   DATA[633,1] := 534.7403;
   DATA[633,2] := 2.0;
   DATA[633,3] := 2.0;
   DATA[633,4] := 262.1764;
   DATA[633,5] := 8.396116;
   DATA[633,6] := 327.7621;
   DATA[633,7] := 2.441675;
   DATA[633,8] := 2.0;
   DATA[633,9] := 2.0;
   DATA[633,10] := 2.0;
   DATA[633,11] := 19.68756;
   DATA[633,12] := 2.209653;
   DATA[633,13] := 985.4845;
   DATA[633,14] := 1.0;
   DATA[633,15] := 2.0;
   DATA[633,16] := 1.0;
   DATA[633,17] := 1.0;
   DATA[633,18] := 1.0;
   DATA[633,19] := 2.0;
   DATA[633,20] := 148.808;
   DATA[633,21] := 155.7806;
   DATA[633,22] := 1.719156;
   DATA[633,23] := 992.5147;
   DATA[633,24] := 2.0;
   DATA[633,25] := 2.0;
   DATA[633,26] := 7.87798;
   DATA[633,27] := 145.0141;
   DATA[633,28] := 263.1377;
   DATA[633,29] := 12.03538;
   DATA[633,30] := 1.731095;
   DATA[633,31] := 1.281542;
   DATA[633,32] := 0.7355248;
   DATA[633,33] := 0.3084265;
   DATA[633,34] := 2.0;
   DATA[633,35] := 250.8972;
   DATA[633,36] := 1.69801;
   DATA[633,37] := 189.6148;
   DATA[633,38] := 0.000128152;
   DATA[633,39] := 1.0;
   DATA[634,0] := 2.641002;
   DATA[634,1] := 534.6618;
   DATA[634,2] := 2.0;
   DATA[634,3] := 2.0;
   DATA[634,4] := 262.1764;
   DATA[634,5] := 8.396116;
   DATA[634,6] := 327.7621;
   DATA[634,7] := 2.44411;
   DATA[634,8] := 2.0;
   DATA[634,9] := 2.0;
   DATA[634,10] := 2.0;
   DATA[634,11] := 19.68756;
   DATA[634,12] := 2.21324;
   DATA[634,13] := 985.4845;
   DATA[634,14] := 1.0;
   DATA[634,15] := 2.0;
   DATA[634,16] := 1.0;
   DATA[634,17] := 1.0;
   DATA[634,18] := 1.0;
   DATA[634,19] := 2.0;
   DATA[634,20] := 148.808;
   DATA[634,21] := 155.7806;
   DATA[634,22] := 1.719156;
   DATA[634,23] := 992.7454;
   DATA[634,24] := 2.0;
   DATA[634,25] := 2.0;
   DATA[634,26] := 7.87798;
   DATA[634,27] := 144.9628;
   DATA[634,28] := 263.1377;
   DATA[634,29] := 12.03538;
   DATA[634,30] := 1.731095;
   DATA[634,31] := 1.281542;
   DATA[634,32] := 0.7355248;
   DATA[634,33] := 0.3080421;
   DATA[634,34] := 2.0;
   DATA[634,35] := 250.8972;
   DATA[634,36] := 1.69801;
   DATA[634,37] := 189.6148;
   DATA[634,38] := 0.000128152;
   DATA[634,39] := 1.0;
   DATA[635,0] := 2.657656;
   DATA[635,1] := 534.1516;
   DATA[635,2] := 2.0;
   DATA[635,3] := 2.0;
   DATA[635,4] := 262.1764;
   DATA[635,5] := 8.396116;
   DATA[635,6] := 327.7621;
   DATA[635,7] := 2.444366;
   DATA[635,8] := 2.0;
   DATA[635,9] := 2.0;
   DATA[635,10] := 2.0;
   DATA[635,11] := 19.68756;
   DATA[635,12] := 2.21324;
   DATA[635,13] := 985.4845;
   DATA[635,14] := 1.0;
   DATA[635,15] := 2.0;
   DATA[635,16] := 1.0;
   DATA[635,17] := 1.0;
   DATA[635,18] := 1.0;
   DATA[635,19] := 2.0;
   DATA[635,20] := 148.808;
   DATA[635,21] := 155.7806;
   DATA[635,22] := 1.717361;
   DATA[635,23] := 992.707;
   DATA[635,24] := 2.0;
   DATA[635,25] := 2.0;
   DATA[635,26] := 7.87798;
   DATA[635,27] := 144.9628;
   DATA[635,28] := 263.1377;
   DATA[635,29] := 12.03538;
   DATA[635,30] := 1.731095;
   DATA[635,31] := 1.282567;
   DATA[635,32] := 0.7355248;
   DATA[635,33] := 0.3066329;
   DATA[635,34] := 2.0;
   DATA[635,35] := 250.8972;
   DATA[635,36] := 1.69801;
   DATA[635,37] := 189.6148;
   DATA[635,38] := 0.000128152;
   DATA[635,39] := 1.0;
   DATA[636,0] := 2.663741;
   DATA[636,1] := 534.23;
   DATA[636,2] := 2.0;
   DATA[636,3] := 2.0;
   DATA[636,4] := 262.1764;
   DATA[636,5] := 8.396116;
   DATA[636,6] := 327.7621;
   DATA[636,7] := 2.444623;
   DATA[636,8] := 2.0;
   DATA[636,9] := 2.0;
   DATA[636,10] := 2.0;
   DATA[636,11] := 19.68756;
   DATA[636,12] := 2.21324;
   DATA[636,13] := 985.3644;
   DATA[636,14] := 1.0;
   DATA[636,15] := 2.0;
   DATA[636,16] := 1.0;
   DATA[636,17] := 1.0;
   DATA[636,18] := 1.0;
   DATA[636,19] := 2.0;
   DATA[636,20] := 148.808;
   DATA[636,21] := 155.7806;
   DATA[636,22] := 1.717361;
   DATA[636,23] := 992.6685;
   DATA[636,24] := 2.0;
   DATA[636,25] := 2.0;
   DATA[636,26] := 7.87798;
   DATA[636,27] := 144.9628;
   DATA[636,28] := 263.1377;
   DATA[636,29] := 12.03538;
   DATA[636,30] := 1.729172;
   DATA[636,31] := 1.289228;
   DATA[636,32] := 0.7355248;
   DATA[636,33] := 0.3081062;
   DATA[636,34] := 2.0;
   DATA[636,35] := 250.8972;
   DATA[636,36] := 1.69801;
   DATA[636,37] := 189.6148;
   DATA[636,38] := 0.000128152;
   DATA[636,39] := 1.0;
   DATA[637,0] := 2.660539;
   DATA[637,1] := 534.5048;
   DATA[637,2] := 2.0;
   DATA[637,3] := 2.0;
   DATA[637,4] := 262.1764;
   DATA[637,5] := 8.396116;
   DATA[637,6] := 327.7621;
   DATA[637,7] := 2.444623;
   DATA[637,8] := 2.0;
   DATA[637,9] := 2.0;
   DATA[637,10] := 2.0;
   DATA[637,11] := 19.67476;
   DATA[637,12] := 2.21324;
   DATA[637,13] := 985.6047;
   DATA[637,14] := 1.0;
   DATA[637,15] := 2.0;
   DATA[637,16] := 1.0;
   DATA[637,17] := 1.0;
   DATA[637,18] := 1.0;
   DATA[637,19] := 2.0;
   DATA[637,20] := 148.808;
   DATA[637,21] := 155.7806;
   DATA[637,22] := 1.717361;
   DATA[637,23] := 992.5916;
   DATA[637,24] := 2.0;
   DATA[637,25] := 2.0;
   DATA[637,26] := 7.87798;
   DATA[637,27] := 144.9628;
   DATA[637,28] := 263.1377;
   DATA[637,29] := 12.03538;
   DATA[637,30] := 1.729172;
   DATA[637,31] := 1.275266;
   DATA[637,32] := 0.7355248;
   DATA[637,33] := 0.3081062;
   DATA[637,34] := 2.0;
   DATA[637,35] := 250.8972;
   DATA[637,36] := 1.69801;
   DATA[637,37] := 189.6148;
   DATA[637,38] := 0.000128152;
   DATA[637,39] := 1.0;
   DATA[638,0] := 2.628511;
   DATA[638,1] := 534.9366;
   DATA[638,2] := 2.0;
   DATA[638,3] := 2.0;
   DATA[638,4] := 262.1764;
   DATA[638,5] := 8.396116;
   DATA[638,6] := 327.7621;
   DATA[638,7] := 2.443341;
   DATA[638,8] := 2.0;
   DATA[638,9] := 2.0;
   DATA[638,10] := 2.0;
   DATA[638,11] := 19.62354;
   DATA[638,12] := 2.211575;
   DATA[638,13] := 985.6848;
   DATA[638,14] := 1.0;
   DATA[638,15] := 2.0;
   DATA[638,16] := 1.0;
   DATA[638,17] := 1.0;
   DATA[638,18] := 1.0;
   DATA[638,19] := 2.0;
   DATA[638,20] := 148.808;
   DATA[638,21] := 155.7806;
   DATA[638,22] := 1.715567;
   DATA[638,23] := 992.5532;
   DATA[638,24] := 2.0;
   DATA[638,25] := 2.0;
   DATA[638,26] := 7.87798;
   DATA[638,27] := 144.9628;
   DATA[638,28] := 263.1377;
   DATA[638,29] := 12.34299;
   DATA[638,30] := 1.729172;
   DATA[638,31] := 1.261304;
   DATA[638,32] := 0.7355248;
   DATA[638,33] := 0.3081062;
   DATA[638,34] := 2.0;
   DATA[638,35] := 250.8972;
   DATA[638,36] := 1.69801;
   DATA[638,37] := 189.6148;
   DATA[638,38] := 0.000128152;
   DATA[638,39] := 1.0;
   DATA[639,0] := 2.622426;
   DATA[639,1] := 535.2114;
   DATA[639,2] := 2.0;
   DATA[639,3] := 2.0;
   DATA[639,4] := 262.1764;
   DATA[639,5] := 8.396116;
   DATA[639,6] := 327.7621;
   DATA[639,7] := 2.443341;
   DATA[639,8] := 2.0;
   DATA[639,9] := 2.0;
   DATA[639,10] := 2.0;
   DATA[639,11] := 19.60753;
   DATA[639,12] := 2.211447;
   DATA[639,13] := 985.8851;
   DATA[639,14] := 1.0;
   DATA[639,15] := 2.0;
   DATA[639,16] := 1.0;
   DATA[639,17] := 1.0;
   DATA[639,18] := 1.0;
   DATA[639,19] := 2.0;
   DATA[639,20] := 148.808;
   DATA[639,21] := 155.7806;
   DATA[639,22] := 1.715567;
   DATA[639,23] := 992.5532;
   DATA[639,24] := 2.0;
   DATA[639,25] := 2.0;
   DATA[639,26] := 7.87798;
   DATA[639,27] := 144.9628;
   DATA[639,28] := 263.1377;
   DATA[639,29] := 12.34299;
   DATA[639,30] := 1.729172;
   DATA[639,31] := 1.261944;
   DATA[639,32] := 0.7355248;
   DATA[639,33] := 0.3081062;
   DATA[639,34] := 2.0;
   DATA[639,35] := 250.8972;
   DATA[639,36] := 1.617916;
   DATA[639,37] := 189.6148;
   DATA[639,38] := 0.000128152;
   DATA[639,39] := 1.0;
   DATA[640,0] := 2.616981;
   DATA[640,1] := 535.2114;
   DATA[640,2] := 2.0;
   DATA[640,3] := 2.0;
   DATA[640,4] := 262.1764;
   DATA[640,5] := 8.395155;
   DATA[640,6] := 327.7621;
   DATA[640,7] := 2.443341;
   DATA[640,8] := 2.0;
   DATA[640,9] := 2.0;
   DATA[640,10] := 2.0;
   DATA[640,11] := 19.57872;
   DATA[640,12] := 2.211447;
   DATA[640,13] := 985.7649;
   DATA[640,14] := 1.0;
   DATA[640,15] := 2.0;
   DATA[640,16] := 1.0;
   DATA[640,17] := 1.0;
   DATA[640,18] := 1.0;
   DATA[640,19] := 2.0;
   DATA[640,20] := 148.808;
   DATA[640,21] := 155.7806;
   DATA[640,22] := 1.715567;
   DATA[640,23] := 992.7839;
   DATA[640,24] := 2.0;
   DATA[640,25] := 2.0;
   DATA[640,26] := 7.87798;
   DATA[640,27] := 144.9628;
   DATA[640,28] := 263.1377;
   DATA[640,29] := 12.34299;
   DATA[640,30] := 1.729172;
   DATA[640,31] := 1.280902;
   DATA[640,32] := 0.7355248;
   DATA[640,33] := 0.3081062;
   DATA[640,34] := 2.0;
   DATA[640,35] := 250.8972;
   DATA[640,36] := 1.617916;
   DATA[640,37] := 189.6148;
   DATA[640,38] := 0.000128152;
   DATA[640,39] := 1.0;
   DATA[641,0] := 2.601287;
   DATA[641,1] := 535.3291;
   DATA[641,2] := 2.0;
   DATA[641,3] := 2.0;
   DATA[641,4] := 262.1764;
   DATA[641,5] := 8.395155;
   DATA[641,6] := 327.7621;
   DATA[641,7] := 2.443341;
   DATA[641,8] := 2.0;
   DATA[641,9] := 2.0;
   DATA[641,10] := 2.0;
   DATA[641,11] := 19.5275;
   DATA[641,12] := 2.211447;
   DATA[641,13] := 986.0052;
   DATA[641,14] := 1.0;
   DATA[641,15] := 2.0;
   DATA[641,16] := 1.0;
   DATA[641,17] := 1.0;
   DATA[641,18] := 1.0;
   DATA[641,19] := 2.0;
   DATA[641,20] := 148.808;
   DATA[641,21] := 155.7806;
   DATA[641,22] := 1.715567;
   DATA[641,23] := 992.8608;
   DATA[641,24] := 2.0;
   DATA[641,25] := 2.0;
   DATA[641,26] := 7.87798;
   DATA[641,27] := 144.9628;
   DATA[641,28] := 263.1377;
   DATA[641,29] := 12.15073;
   DATA[641,30] := 1.729172;
   DATA[641,31] := 1.28167;
   DATA[641,32] := 0.7355248;
   DATA[641,33] := 0.3081062;
   DATA[641,34] := 2.0;
   DATA[641,35] := 250.8972;
   DATA[641,36] := 1.617916;
   DATA[641,37] := 189.6148;
   DATA[641,38] := 0.000128152;
   DATA[641,39] := 1.0;
   DATA[642,0] := 2.585914;
   DATA[642,1] := 535.4469;
   DATA[642,2] := 2.0;
   DATA[642,3] := 2.0;
   DATA[642,4] := 262.1764;
   DATA[642,5] := 8.395155;
   DATA[642,6] := 327.7621;
   DATA[642,7] := 2.440393;
   DATA[642,8] := 2.0;
   DATA[642,9] := 2.0;
   DATA[642,10] := 2.0;
   DATA[642,11] := 19.5275;
   DATA[642,12] := 2.211447;
   DATA[642,13] := 986.0853;
   DATA[642,14] := 1.0;
   DATA[642,15] := 2.0;
   DATA[642,16] := 1.0;
   DATA[642,17] := 1.0;
   DATA[642,18] := 1.0;
   DATA[642,19] := 2.0;
   DATA[642,20] := 148.808;
   DATA[642,21] := 155.7806;
   DATA[642,22] := 1.715567;
   DATA[642,23] := 992.9761;
   DATA[642,24] := 2.0;
   DATA[642,25] := 2.0;
   DATA[642,26] := 7.878942;
   DATA[642,27] := 144.9628;
   DATA[642,28] := 263.1377;
   DATA[642,29] := 12.03538;
   DATA[642,30] := 1.729172;
   DATA[642,31] := 1.28167;
   DATA[642,32] := 0.7339884;
   DATA[642,33] := 0.3084905;
   DATA[642,34] := 2.0;
   DATA[642,35] := 250.8972;
   DATA[642,36] := 1.617916;
   DATA[642,37] := 189.6148;
   DATA[642,38] := 0.000128152;
   DATA[642,39] := 1.0;
   DATA[643,0] := 2.564456;
   DATA[643,1] := 535.8394;
   DATA[643,2] := 2.0;
   DATA[643,3] := 2.0;
   DATA[643,4] := 262.1764;
   DATA[643,5] := 8.395155;
   DATA[643,6] := 327.7621;
   DATA[643,7] := 2.439753;
   DATA[643,8] := 2.0;
   DATA[643,9] := 2.0;
   DATA[643,10] := 2.0;
   DATA[643,11] := 19.5275;
   DATA[643,12] := 2.211447;
   DATA[643,13] := 986.0853;
   DATA[643,14] := 1.0;
   DATA[643,15] := 2.0;
   DATA[643,16] := 1.0;
   DATA[643,17] := 1.0;
   DATA[643,18] := 1.0;
   DATA[643,19] := 2.0;
   DATA[643,20] := 148.808;
   DATA[643,21] := 155.7806;
   DATA[643,22] := 1.715567;
   DATA[643,23] := 993.053;
   DATA[643,24] := 2.0;
   DATA[643,25] := 2.0;
   DATA[643,26] := 7.878942;
   DATA[643,27] := 144.9628;
   DATA[643,28] := 263.1377;
   DATA[643,29] := 12.03538;
   DATA[643,30] := 1.730838;
   DATA[643,31] := 1.277956;
   DATA[643,32] := 0.7339884;
   DATA[643,33] := 0.3084905;
   DATA[643,34] := 2.0;
   DATA[643,35] := 250.8972;
   DATA[643,36] := 1.617916;
   DATA[643,37] := 189.6148;
   DATA[643,38] := 0.000128152;
   DATA[643,39] := 1.0;
   DATA[644,0] := 2.548762;
   DATA[644,1] := 535.6431;
   DATA[644,2] := 2.0;
   DATA[644,3] := 2.0;
   DATA[644,4] := 262.1764;
   DATA[644,5] := 8.395155;
   DATA[644,6] := 327.7621;
   DATA[644,7] := 2.439753;
   DATA[644,8] := 2.0;
   DATA[644,9] := 2.0;
   DATA[644,10] := 2.0;
   DATA[644,11] := 19.59793;
   DATA[644,12] := 2.210166;
   DATA[644,13] := 986.2856;
   DATA[644,14] := 1.0;
   DATA[644,15] := 2.0;
   DATA[644,16] := 1.0;
   DATA[644,17] := 1.0;
   DATA[644,18] := 1.0;
   DATA[644,19] := 2.0;
   DATA[644,20] := 148.808;
   DATA[644,21] := 155.7806;
   DATA[644,22] := 1.715567;
   DATA[644,23] := 993.0915;
   DATA[644,24] := 2.0;
   DATA[644,25] := 2.0;
   DATA[644,26] := 7.878942;
   DATA[644,27] := 144.9628;
   DATA[644,28] := 263.1697;
   DATA[644,29] := 12.03538;
   DATA[644,30] := 1.730838;
   DATA[644,31] := 1.275266;
   DATA[644,32] := 0.7360369;
   DATA[644,33] := 0.3084905;
   DATA[644,34] := 2.0;
   DATA[644,35] := 250.8011;
   DATA[644,36] := 1.762086;
   DATA[644,37] := 189.5668;
   DATA[644,38] := 0.000128152;
   DATA[644,39] := 1.0;
   DATA[645,0] := 2.533068;
   DATA[645,1] := 535.2506;
   DATA[645,2] := 2.0;
   DATA[645,3] := 2.0;
   DATA[645,4] := 262.1764;
   DATA[645,5] := 8.395155;
   DATA[645,6] := 327.7621;
   DATA[645,7] := 2.439753;
   DATA[645,8] := 2.0;
   DATA[645,9] := 2.0;
   DATA[645,10] := 2.0;
   DATA[645,11] := 19.62674;
   DATA[645,12] := 2.210166;
   DATA[645,13] := 986.6461;
   DATA[645,14] := 1.0;
   DATA[645,15] := 2.0;
   DATA[645,16] := 1.0;
   DATA[645,17] := 1.0;
   DATA[645,18] := 1.0;
   DATA[645,19] := 2.0;
   DATA[645,20] := 148.808;
   DATA[645,21] := 155.7806;
   DATA[645,22] := 1.714798;
   DATA[645,23] := 992.9761;
   DATA[645,24] := 2.0;
   DATA[645,25] := 2.0;
   DATA[645,26] := 7.878942;
   DATA[645,27] := 144.9628;
   DATA[645,28] := 263.4261;
   DATA[645,29] := 12.03538;
   DATA[645,30] := 1.730838;
   DATA[645,31] := 1.289484;
   DATA[645,32] := 0.7360369;
   DATA[645,33] := 0.3074016;
   DATA[645,34] := 2.0;
   DATA[645,35] := 250.6569;
   DATA[645,36] := 1.762086;
   DATA[645,37] := 189.5347;
   DATA[645,38] := 0.000128152;
   DATA[645,39] := 1.0;
   DATA[646,0] := 2.517695;
   DATA[646,1] := 534.8973;
   DATA[646,2] := 2.0;
   DATA[646,3] := 2.0;
   DATA[646,4] := 262.1764;
   DATA[646,5] := 8.395155;
   DATA[646,6] := 327.7621;
   DATA[646,7] := 2.439753;
   DATA[646,8] := 2.0;
   DATA[646,9] := 2.0;
   DATA[646,10] := 2.0;
   DATA[646,11] := 19.62674;
   DATA[646,12] := 2.210166;
   DATA[646,13] := 987.0466;
   DATA[646,14] := 1.0;
   DATA[646,15] := 2.0;
   DATA[646,16] := 1.0;
   DATA[646,17] := 1.0;
   DATA[646,18] := 1.0;
   DATA[646,19] := 2.0;
   DATA[646,20] := 148.808;
   DATA[646,21] := 155.7806;
   DATA[646,22] := 1.714542;
   DATA[646,23] := 993.053;
   DATA[646,24] := 2.0;
   DATA[646,25] := 2.0;
   DATA[646,26] := 7.878942;
   DATA[646,27] := 145.1166;
   DATA[646,28] := 263.4261;
   DATA[646,29] := 12.03538;
   DATA[646,30] := 1.727634;
   DATA[646,31] := 1.300756;
   DATA[646,32] := 0.7360369;
   DATA[646,33] := 0.3068251;
   DATA[646,34] := 2.0;
   DATA[646,35] := 250.6569;
   DATA[646,36] := 1.762086;
   DATA[646,37] := 189.5027;
   DATA[646,38] := 0.000128152;
   DATA[646,39] := 1.0;
   DATA[647,0] := 2.498799;
   DATA[647,1] := 534.6226;
   DATA[647,2] := 2.0;
   DATA[647,3] := 2.0;
   DATA[647,4] := 262.1764;
   DATA[647,5] := 8.395155;
   DATA[647,6] := 327.7621;
   DATA[647,7] := 2.439753;
   DATA[647,8] := 2.0;
   DATA[647,9] := 2.0;
   DATA[647,10] := 2.0;
   DATA[647,11] := 19.62674;
   DATA[647,12] := 2.211447;
   DATA[647,13] := 987.4471;
   DATA[647,14] := 1.0;
   DATA[647,15] := 2.0;
   DATA[647,16] := 1.0;
   DATA[647,17] := 1.0;
   DATA[647,18] := 1.0;
   DATA[647,19] := 2.0;
   DATA[647,20] := 148.808;
   DATA[647,21] := 155.7806;
   DATA[647,22] := 1.714542;
   DATA[647,23] := 992.8992;
   DATA[647,24] := 2.0;
   DATA[647,25] := 2.0;
   DATA[647,26] := 7.878942;
   DATA[647,27] := 145.1166;
   DATA[647,28] := 263.4261;
   DATA[647,29] := 12.03538;
   DATA[647,30] := 1.727634;
   DATA[647,31] := 1.297554;
   DATA[647,32] := 0.7360369;
   DATA[647,33] := 0.3068251;
   DATA[647,34] := 2.0;
   DATA[647,35] := 250.6569;
   DATA[647,36] := 1.601897;
   DATA[647,37] := 189.3745;
   DATA[647,38] := 0.000128152;
   DATA[647,39] := 1.0;
   DATA[648,0] := 2.483426;
   DATA[648,1] := 534.3085;
   DATA[648,2] := 2.0;
   DATA[648,3] := 2.0;
   DATA[648,4] := 262.1764;
   DATA[648,5] := 8.395155;
   DATA[648,6] := 327.7621;
   DATA[648,7] := 2.439753;
   DATA[648,8] := 2.0;
   DATA[648,9] := 2.0;
   DATA[648,10] := 2.0;
   DATA[648,11] := 19.66835;
   DATA[648,12] := 2.211447;
   DATA[648,13] := 987.0867;
   DATA[648,14] := 1.0;
   DATA[648,15] := 2.0;
   DATA[648,16] := 1.0;
   DATA[648,17] := 1.0;
   DATA[648,18] := 1.0;
   DATA[648,19] := 2.0;
   DATA[648,20] := 148.808;
   DATA[648,21] := 155.7806;
   DATA[648,22] := 1.715824;
   DATA[648,23] := 993.2453;
   DATA[648,24] := 2.0;
   DATA[648,25] := 2.0;
   DATA[648,26] := 7.878942;
   DATA[648,27] := 145.1166;
   DATA[648,28] := 263.4261;
   DATA[648,29] := 12.03538;
   DATA[648,30] := 1.727634;
   DATA[648,31] := 1.291918;
   DATA[648,32] := 0.7346286;
   DATA[648,33] := 0.3068251;
   DATA[648,34] := 2.0;
   DATA[648,35] := 250.6569;
   DATA[648,36] := 1.601897;
   DATA[648,37] := 189.3745;
   DATA[648,38] := 0.000128152;
   DATA[648,39] := 1.0;
   DATA[649,0] := 2.463248;
   DATA[649,1] := 534.6226;
   DATA[649,2] := 2.0;
   DATA[649,3] := 2.0;
   DATA[649,4] := 262.1764;
   DATA[649,5] := 8.395155;
   DATA[649,6] := 327.7621;
   DATA[649,7] := 2.439753;
   DATA[649,8] := 2.0;
   DATA[649,9] := 2.0;
   DATA[649,10] := 2.0;
   DATA[649,11] := 19.57552;
   DATA[649,12] := 2.211447;
   DATA[649,13] := 987.2068;
   DATA[649,14] := 1.0;
   DATA[649,15] := 2.0;
   DATA[649,16] := 1.0;
   DATA[649,17] := 1.0;
   DATA[649,18] := 1.0;
   DATA[649,19] := 2.0;
   DATA[649,20] := 148.808;
   DATA[649,21] := 155.7806;
   DATA[649,22] := 1.716849;
   DATA[649,23] := 993.2453;
   DATA[649,24] := 2.0;
   DATA[649,25] := 2.0;
   DATA[649,26] := 7.878942;
   DATA[649,27] := 145.1166;
   DATA[649,28] := 263.1697;
   DATA[649,29] := 12.03538;
   DATA[649,30] := 1.727634;
   DATA[649,31] := 1.281927;
   DATA[649,32] := 0.7346286;
   DATA[649,33] := 0.3066329;
   DATA[649,34] := 2.0;
   DATA[649,35] := 250.6569;
   DATA[649,36] := 1.601897;
   DATA[649,37] := 189.3745;
   DATA[649,38] := 0.000128152;
   DATA[649,39] := 1.0;
   DATA[650,0] := 2.463248;
   DATA[650,1] := 534.6226;
   DATA[650,2] := 2.0;
   DATA[650,3] := 2.0;
   DATA[650,4] := 262.1764;
   DATA[650,5] := 8.395155;
   DATA[650,6] := 327.7621;
   DATA[650,7] := 2.439753;
   DATA[650,8] := 2.0;
   DATA[650,9] := 2.0;
   DATA[650,10] := 2.0;
   DATA[650,11] := 19.57552;
   DATA[650,12] := 2.211447;
   DATA[650,13] := 987.2068;
   DATA[650,14] := 1.0;
   DATA[650,15] := 2.0;
   DATA[650,16] := 1.0;
   DATA[650,17] := 1.0;
   DATA[650,18] := 1.0;
   DATA[650,19] := 2.0;
   DATA[650,20] := 148.808;
   DATA[650,21] := 155.7806;
   DATA[650,22] := 1.716849;
   DATA[650,23] := 993.2453;
   DATA[650,24] := 2.0;
   DATA[650,25] := 2.0;
   DATA[650,26] := 7.878942;
   DATA[650,27] := 145.1166;
   DATA[650,28] := 263.1697;
   DATA[650,29] := 12.03538;
   DATA[650,30] := 1.727634;
   DATA[650,31] := 1.281927;
   DATA[650,32] := 0.7346286;
   DATA[650,33] := 0.3066329;
   DATA[650,34] := 2.0;
   DATA[650,35] := 250.6569;
   DATA[650,36] := 1.601897;
   DATA[650,37] := 189.3745;
   DATA[650,38] := 0.000128152;
   DATA[650,39] := 1.0;
   DATA[651,0] := 2.447234;
   DATA[651,1] := 534.701;
   DATA[651,2] := 2.0;
   DATA[651,3] := 2.0;
   DATA[651,4] := 262.1764;
   DATA[651,5] := 8.395155;
   DATA[651,6] := 327.7621;
   DATA[651,7] := 2.439753;
   DATA[651,8] := 2.0;
   DATA[651,9] := 2.0;
   DATA[651,10] := 2.0;
   DATA[651,11] := 19.57552;
   DATA[651,12] := 2.212856;
   DATA[651,13] := 987.0065;
   DATA[651,14] := 1.0;
   DATA[651,15] := 2.0;
   DATA[651,16] := 1.0;
   DATA[651,17] := 1.0;
   DATA[651,18] := 1.0;
   DATA[651,19] := 2.0;
   DATA[651,20] := 148.808;
   DATA[651,21] := 155.7806;
   DATA[651,22] := 1.717361;
   DATA[651,23] := 993.1684;
   DATA[651,24] := 2.0;
   DATA[651,25] := 2.0;
   DATA[651,26] := 7.878942;
   DATA[651,27] := 145.1166;
   DATA[651,28] := 263.1697;
   DATA[651,29] := 12.03538;
   DATA[651,30] := 1.727634;
   DATA[651,31] := 1.281158;
   DATA[651,32] := 0.7346286;
   DATA[651,33] := 0.3066329;
   DATA[651,34] := 2.0;
   DATA[651,35] := 250.8331;
   DATA[651,36] := 1.601897;
   DATA[651,37] := 189.6629;
   DATA[651,38] := 0.000128152;
   DATA[651,39] := 1.0;
   DATA[652,0] := 2.431861;
   DATA[652,1] := 535.9179;
   DATA[652,2] := 2.0;
   DATA[652,3] := 2.0;
   DATA[652,4] := 262.1764;
   DATA[652,5] := 8.395155;
   DATA[652,6] := 327.7621;
   DATA[652,7] := 2.44206;
   DATA[652,8] := 2.0;
   DATA[652,9] := 2.0;
   DATA[652,10] := 2.0;
   DATA[652,11] := 19.57552;
   DATA[652,12] := 2.212856;
   DATA[652,13] := 987.0466;
   DATA[652,14] := 1.0;
   DATA[652,15] := 2.0;
   DATA[652,16] := 1.0;
   DATA[652,17] := 1.0;
   DATA[652,18] := 1.0;
   DATA[652,19] := 2.0;
   DATA[652,20] := 148.808;
   DATA[652,21] := 155.7806;
   DATA[652,22] := 1.719284;
   DATA[652,23] := 993.3607;
   DATA[652,24] := 2.0;
   DATA[652,25] := 2.0;
   DATA[652,26] := 7.878942;
   DATA[652,27] := 145.1166;
   DATA[652,28] := 263.1697;
   DATA[652,29] := 12.03538;
   DATA[652,30] := 1.725968;
   DATA[652,31] := 1.289356;
   DATA[652,32] := 0.7361649;
   DATA[652,33] := 0.3066329;
   DATA[652,34] := 2.0;
   DATA[652,35] := 250.8331;
   DATA[652,36] := 1.601897;
   DATA[652,37] := 189.6629;
   DATA[652,38] := 0.000128152;
   DATA[652,39] := 1.0;
   DATA[653,0] := 2.428979;
   DATA[653,1] := 537.017;
   DATA[653,2] := 2.0;
   DATA[653,3] := 2.0;
   DATA[653,4] := 262.1764;
   DATA[653,5] := 8.395155;
   DATA[653,6] := 327.7621;
   DATA[653,7] := 2.44206;
   DATA[653,8] := 2.0;
   DATA[653,9] := 2.0;
   DATA[653,10] := 2.0;
   DATA[653,11] := 19.67155;
   DATA[653,12] := 2.212856;
   DATA[653,13] := 987.9678;
   DATA[653,14] := 1.0;
   DATA[653,15] := 2.0;
   DATA[653,16] := 1.0;
   DATA[653,17] := 1.0;
   DATA[653,18] := 1.0;
   DATA[653,19] := 2.0;
   DATA[653,20] := 148.808;
   DATA[653,21] := 155.7806;
   DATA[653,22] := 1.719412;
   DATA[653,23] := 993.8605;
   DATA[653,24] := 2.0;
   DATA[653,25] := 2.0;
   DATA[653,26] := 7.878942;
   DATA[653,27] := 145.0141;
   DATA[653,28] := 263.1697;
   DATA[653,29] := 12.03538;
   DATA[653,30] := 1.725968;
   DATA[653,31] := 1.296273;
   DATA[653,32] := 0.7361649;
   DATA[653,33] := 0.3066329;
   DATA[653,34] := 2.0;
   DATA[653,35] := 250.9613;
   DATA[653,36] := 1.601897;
   DATA[653,37] := 189.6629;
   DATA[653,38] := 0.000128152;
   DATA[653,39] := 1.0;
   DATA[654,0] := 2.431861;
   DATA[654,1] := 537.488;
   DATA[654,2] := 2.0;
   DATA[654,3] := 2.0;
   DATA[654,4] := 262.1764;
   DATA[654,5] := 8.395155;
   DATA[654,6] := 327.7621;
   DATA[654,7] := 2.44206;
   DATA[654,8] := 2.0;
   DATA[654,9] := 2.0;
   DATA[654,10] := 2.0;
   DATA[654,11] := 19.67155;
   DATA[654,12] := 2.212856;
   DATA[654,13] := 987.7676;
   DATA[654,14] := 1.0;
   DATA[654,15] := 2.0;
   DATA[654,16] := 1.0;
   DATA[654,17] := 1.0;
   DATA[654,18] := 1.0;
   DATA[654,19] := 2.0;
   DATA[654,20] := 148.808;
   DATA[654,21] := 155.7806;
   DATA[654,22] := 1.719412;
   DATA[654,23] := 994.1297;
   DATA[654,24] := 2.0;
   DATA[654,25] := 2.0;
   DATA[654,26] := 7.878942;
   DATA[654,27] := 144.9628;
   DATA[654,28] := 263.1697;
   DATA[654,29] := 12.03538;
   DATA[654,30] := 1.729557;
   DATA[654,31] := 1.308825;
   DATA[654,32] := 0.7361649;
   DATA[654,33] := 0.3066329;
   DATA[654,34] := 2.0;
   DATA[654,35] := 250.9613;
   DATA[654,36] := 1.601897;
   DATA[654,37] := 189.6629;
   DATA[654,38] := 0.000128152;
   DATA[654,39] := 1.0;
   DATA[655,0] := 2.475419;
   DATA[655,1] := 537.8806;
   DATA[655,2] := 2.0;
   DATA[655,3] := 2.0;
   DATA[655,4] := 262.1764;
   DATA[655,5] := 8.395155;
   DATA[655,6] := 327.7621;
   DATA[655,7] := 2.44206;
   DATA[655,8] := 2.0;
   DATA[655,9] := 2.0;
   DATA[655,10] := 2.0;
   DATA[655,11] := 19.67155;
   DATA[655,12] := 2.21119;
   DATA[655,13] := 987.8878;
   DATA[655,14] := 1.0;
   DATA[655,15] := 2.0;
   DATA[655,16] := 1.0;
   DATA[655,17] := 1.0;
   DATA[655,18] := 1.0;
   DATA[655,19] := 2.0;
   DATA[655,20] := 148.808;
   DATA[655,21] := 155.7806;
   DATA[655,22] := 1.719412;
   DATA[655,23] := 994.5142;
   DATA[655,24] := 2.0;
   DATA[655,25] := 2.0;
   DATA[655,26] := 7.878942;
   DATA[655,27] := 144.9628;
   DATA[655,28] := 263.1697;
   DATA[655,29] := 12.03538;
   DATA[655,30] := 1.730454;
   DATA[655,31] := 1.305495;
   DATA[655,32] := 0.7342445;
   DATA[655,33] := 0.3066329;
   DATA[655,34] := 2.0;
   DATA[655,35] := 251.1215;
   DATA[655,36] := 1.746067;
   DATA[655,37] := 189.6629;
   DATA[655,38] := 0.000128152;
   DATA[655,39] := 1.0;
   DATA[656,0] := 2.526022;
   DATA[656,1] := 538.1553;
   DATA[656,2] := 2.0;
   DATA[656,3] := 2.0;
   DATA[656,4] := 262.1764;
   DATA[656,5] := 8.395155;
   DATA[656,6] := 327.7621;
   DATA[656,7] := 2.44206;
   DATA[656,8] := 2.0;
   DATA[656,9] := 2.0;
   DATA[656,10] := 2.0;
   DATA[656,11] := 19.62994;
   DATA[656,12] := 2.210806;
   DATA[656,13] := 988.048;
   DATA[656,14] := 1.0;
   DATA[656,15] := 2.0;
   DATA[656,16] := 1.0;
   DATA[656,17] := 1.0;
   DATA[656,18] := 1.0;
   DATA[656,19] := 2.0;
   DATA[656,20] := 148.808;
   DATA[656,21] := 155.7806;
   DATA[656,22] := 1.719412;
   DATA[656,23] := 994.5142;
   DATA[656,24] := 2.0;
   DATA[656,25] := 2.0;
   DATA[656,26] := 7.878942;
   DATA[656,27] := 144.9628;
   DATA[656,28] := 263.1697;
   DATA[656,29] := 12.03538;
   DATA[656,30] := 1.73071;
   DATA[656,31] := 1.311387;
   DATA[656,32] := 0.7342445;
   DATA[656,33] := 0.3066329;
   DATA[656,34] := 2.0;
   DATA[656,35] := 251.1375;
   DATA[656,36] := 1.746067;
   DATA[656,37] := 189.759;
   DATA[656,38] := 0.000128152;
   DATA[656,39] := 1.0;
   DATA[657,0] := 2.556449;
   DATA[657,1] := 537.8413;
   DATA[657,2] := 2.0;
   DATA[657,3] := 2.0;
   DATA[657,4] := 262.1764;
   DATA[657,5] := 8.395155;
   DATA[657,6] := 327.7621;
   DATA[657,7] := 2.44206;
   DATA[657,8] := 2.0;
   DATA[657,9] := 2.0;
   DATA[657,10] := 2.0;
   DATA[657,11] := 19.62994;
   DATA[657,12] := 2.210806;
   DATA[657,13] := 988.2883;
   DATA[657,14] := 1.0;
   DATA[657,15] := 2.0;
   DATA[657,16] := 1.0;
   DATA[657,17] := 1.0;
   DATA[657,18] := 1.0;
   DATA[657,19] := 2.0;
   DATA[657,20] := 148.808;
   DATA[657,21] := 155.7806;
   DATA[657,22] := 1.719412;
   DATA[657,23] := 995.0141;
   DATA[657,24] := 2.0;
   DATA[657,25] := 2.0;
   DATA[657,26] := 7.878942;
   DATA[657,27] := 144.9628;
   DATA[657,28] := 263.1697;
   DATA[657,29] := 12.07383;
   DATA[657,30] := 1.73071;
   DATA[657,31] := 1.307929;
   DATA[657,32] := 0.7342445;
   DATA[657,33] := 0.3066329;
   DATA[657,34] := 2.0;
   DATA[657,35] := 251.3779;
   DATA[657,36] := 1.746067;
   DATA[657,37] := 189.8071;
   DATA[657,38] := 0.000128152;
   DATA[657,39] := 1.0;
   DATA[658,0] := 2.597764;
   DATA[658,1] := 537.6058;
   DATA[658,2] := 2.0;
   DATA[658,3] := 2.0;
   DATA[658,4] := 262.1764;
   DATA[658,5] := 8.395155;
   DATA[658,6] := 327.7621;
   DATA[658,7] := 2.44206;
   DATA[658,8] := 2.0;
   DATA[658,9] := 2.0;
   DATA[658,10] := 2.0;
   DATA[658,11] := 19.62994;
   DATA[658,12] := 2.210806;
   DATA[658,13] := 988.4084;
   DATA[658,14] := 1.0;
   DATA[658,15] := 2.0;
   DATA[658,16] := 1.0;
   DATA[658,17] := 1.0;
   DATA[658,18] := 1.0;
   DATA[658,19] := 2.0;
   DATA[658,20] := 148.808;
   DATA[658,21] := 155.7806;
   DATA[658,22] := 1.719412;
   DATA[658,23] := 995.0526;
   DATA[658,24] := 2.0;
   DATA[658,25] := 2.0;
   DATA[658,26] := 7.878942;
   DATA[658,27] := 144.9628;
   DATA[658,28] := 263.1697;
   DATA[658,29] := 12.07383;
   DATA[658,30] := 1.73212;
   DATA[658,31] := 1.30178;
   DATA[658,32] := 0.7352687;
   DATA[658,33] := 0.3066329;
   DATA[658,34] := 2.0;
   DATA[658,35] := 251.3779;
   DATA[658,36] := 1.746067;
   DATA[658,37] := 189.9353;
   DATA[658,38] := 0.000128152;
   DATA[658,39] := 1.0;
   DATA[659,0] := 2.626589;
   DATA[659,1] := 537.4095;
   DATA[659,2] := 2.0;
   DATA[659,3] := 2.0;
   DATA[659,4] := 262.1764;
   DATA[659,5] := 8.395155;
   DATA[659,6] := 327.7621;
   DATA[659,7] := 2.440906;
   DATA[659,8] := 2.0;
   DATA[659,9] := 2.0;
   DATA[659,10] := 2.0;
   DATA[659,11] := 19.62994;
   DATA[659,12] := 2.210806;
   DATA[659,13] := 988.4485;
   DATA[659,14] := 1.0;
   DATA[659,15] := 2.0;
   DATA[659,16] := 1.0;
   DATA[659,17] := 1.0;
   DATA[659,18] := 1.0;
   DATA[659,19] := 2.0;
   DATA[659,20] := 148.808;
   DATA[659,21] := 155.7806;
   DATA[659,22] := 1.719412;
   DATA[659,23] := 995.3986;
   DATA[659,24] := 2.0;
   DATA[659,25] := 2.0;
   DATA[659,26] := 7.878942;
   DATA[659,27] := 144.9628;
   DATA[659,28] := 263.2658;
   DATA[659,29] := 12.07383;
   DATA[659,30] := 1.73212;
   DATA[659,31] := 1.293711;
   DATA[659,32] := 0.7359089;
   DATA[659,33] := 0.3066329;
   DATA[659,34] := 2.0;
   DATA[659,35] := 251.3779;
   DATA[659,36] := 1.746067;
   DATA[659,37] := 189.9353;
   DATA[659,38] := 0.000128152;
   DATA[659,39] := 1.0;
   DATA[660,0] := 2.657016;
   DATA[660,1] := 537.3702;
   DATA[660,2] := 2.0;
   DATA[660,3] := 2.0;
   DATA[660,4] := 262.1764;
   DATA[660,5] := 8.395155;
   DATA[660,6] := 327.7621;
   DATA[660,7] := 2.440906;
   DATA[660,8] := 2.0;
   DATA[660,9] := 2.0;
   DATA[660,10] := 2.0;
   DATA[660,11] := 19.62994;
   DATA[660,12] := 2.210806;
   DATA[660,13] := 988.2883;
   DATA[660,14] := 1.0;
   DATA[660,15] := 2.0;
   DATA[660,16] := 1.0;
   DATA[660,17] := 1.0;
   DATA[660,18] := 1.0;
   DATA[660,19] := 2.0;
   DATA[660,20] := 148.808;
   DATA[660,21] := 155.7806;
   DATA[660,22] := 1.72159;
   DATA[660,23] := 995.4755;
   DATA[660,24] := 2.0;
   DATA[660,25] := 2.0;
   DATA[660,26] := 7.878942;
   DATA[660,27] := 144.9628;
   DATA[660,28] := 263.362;
   DATA[660,29] := 12.07383;
   DATA[660,30] := 1.73212;
   DATA[660,31] := 1.28372;
   DATA[660,32] := 0.7359089;
   DATA[660,33] := 0.3066329;
   DATA[660,34] := 2.0;
   DATA[660,35] := 251.2016;
   DATA[660,36] := 1.746067;
   DATA[660,37] := 189.9353;
   DATA[660,38] := 0.000128152;
   DATA[660,39] := 1.0;
   DATA[661,0] := 2.667585;
   DATA[661,1] := 537.0562;
   DATA[661,2] := 2.0;
   DATA[661,3] := 2.0;
   DATA[661,4] := 262.1764;
   DATA[661,5] := 8.395155;
   DATA[661,6] := 327.7621;
   DATA[661,7] := 2.440906;
   DATA[661,8] := 2.0;
   DATA[661,9] := 2.0;
   DATA[661,10] := 2.0;
   DATA[661,11] := 19.65555;
   DATA[661,12] := 2.209525;
   DATA[661,13] := 988.5687;
   DATA[661,14] := 1.0;
   DATA[661,15] := 2.0;
   DATA[661,16] := 1.0;
   DATA[661,17] := 1.0;
   DATA[661,18] := 1.0;
   DATA[661,19] := 2.0;
   DATA[661,20] := 148.808;
   DATA[661,21] := 155.7806;
   DATA[661,22] := 1.721975;
   DATA[661,23] := 995.6293;
   DATA[661,24] := 2.0;
   DATA[661,25] := 2.0;
   DATA[661,26] := 7.878942;
   DATA[661,27] := 144.9628;
   DATA[661,28] := 263.362;
   DATA[661,29] := 12.07383;
   DATA[661,30] := 1.73212;
   DATA[661,31] := 1.272192;
   DATA[661,32] := 0.7359089;
   DATA[661,33] := 0.3066329;
   DATA[661,34] := 2.0;
   DATA[661,35] := 251.0574;
   DATA[661,36] := 1.746067;
   DATA[661,37] := 189.9353;
   DATA[661,38] := 0.000128152;
   DATA[661,39] := 1.0;
   DATA[662,0] := 2.657976;
   DATA[662,1] := 537.0955;
   DATA[662,2] := 2.0;
   DATA[662,3] := 2.0;
   DATA[662,4] := 262.1764;
   DATA[662,5] := 8.395155;
   DATA[662,6] := 327.7621;
   DATA[662,7] := 2.443725;
   DATA[662,8] := 2.0;
   DATA[662,9] := 2.0;
   DATA[662,10] := 2.0;
   DATA[662,11] := 19.65555;
   DATA[662,12] := 2.209525;
   DATA[662,13] := 988.4485;
   DATA[662,14] := 1.0;
   DATA[662,15] := 2.0;
   DATA[662,16] := 1.0;
   DATA[662,17] := 1.0;
   DATA[662,18] := 1.0;
   DATA[662,19] := 2.0;
   DATA[662,20] := 148.808;
   DATA[662,21] := 155.7806;
   DATA[662,22] := 1.721975;
   DATA[662,23] := 996.0139;
   DATA[662,24] := 2.0;
   DATA[662,25] := 2.0;
   DATA[662,26] := 7.878942;
   DATA[662,27] := 144.9628;
   DATA[662,28] := 263.362;
   DATA[662,29] := 12.07383;
   DATA[662,30] := 1.73212;
   DATA[662,31] := 1.271295;
   DATA[662,32] := 0.7359089;
   DATA[662,33] := 0.3066329;
   DATA[662,34] := 2.0;
   DATA[662,35] := 251.0574;
   DATA[662,36] := 1.746067;
   DATA[662,37] := 189.9353;
   DATA[662,38] := 0.000128152;
   DATA[662,39] := 1.0;
   DATA[663,0] := 2.631393;
   DATA[663,1] := 537.2133;
   DATA[663,2] := 2.0;
   DATA[663,3] := 2.0;
   DATA[663,4] := 262.1764;
   DATA[663,5] := 8.395155;
   DATA[663,6] := 327.7621;
   DATA[663,7] := 2.444366;
   DATA[663,8] := 2.0;
   DATA[663,9] := 2.0;
   DATA[663,10] := 2.0;
   DATA[663,11] := 19.65555;
   DATA[663,12] := 2.213368;
   DATA[663,13] := 988.048;
   DATA[663,14] := 1.0;
   DATA[663,15] := 2.0;
   DATA[663,16] := 1.0;
   DATA[663,17] := 1.0;
   DATA[663,18] := 1.0;
   DATA[663,19] := 2.0;
   DATA[663,20] := 148.808;
   DATA[663,21] := 155.7806;
   DATA[663,22] := 1.720565;
   DATA[663,23] := 995.9754;
   DATA[663,24] := 2.0;
   DATA[663,25] := 2.0;
   DATA[663,26] := 7.878942;
   DATA[663,27] := 144.9628;
   DATA[663,28] := 263.362;
   DATA[663,29] := 12.07383;
   DATA[663,30] := 1.73212;
   DATA[663,31] := 1.262073;
   DATA[663,32] := 0.7357808;
   DATA[663,33] := 0.3066329;
   DATA[663,34] := 2.0;
   DATA[663,35] := 251.0574;
   DATA[663,36] := 1.746067;
   DATA[663,37] := 189.759;
   DATA[663,38] := 0.000128152;
   DATA[663,39] := 1.0;
   DATA[664,0] := 2.620824;
   DATA[664,1] := 537.0955;
   DATA[664,2] := 2.0;
   DATA[664,3] := 2.0;
   DATA[664,4] := 262.1764;
   DATA[664,5] := 8.395155;
   DATA[664,6] := 327.7621;
   DATA[664,7] := 2.445007;
   DATA[664,8] := 2.0;
   DATA[664,9] := 2.0;
   DATA[664,10] := 2.0;
   DATA[664,11] := 19.70357;
   DATA[664,12] := 2.211831;
   DATA[664,13] := 987.8878;
   DATA[664,14] := 1.0;
   DATA[664,15] := 2.0;
   DATA[664,16] := 1.0;
   DATA[664,17] := 1.0;
   DATA[664,18] := 1.0;
   DATA[664,19] := 2.0;
   DATA[664,20] := 148.808;
   DATA[664,21] := 155.6524;
   DATA[664,22] := 1.719027;
   DATA[664,23] := 996.2446;
   DATA[664,24] := 2.0;
   DATA[664,25] := 2.0;
   DATA[664,26] := 7.878942;
   DATA[664,27] := 144.9628;
   DATA[664,28] := 263.362;
   DATA[664,29] := 12.07383;
   DATA[664,30] := 1.73212;
   DATA[664,31] := 1.254771;
   DATA[664,32] := 0.7357808;
   DATA[664,33] := 0.3066329;
   DATA[664,34] := 2.0;
   DATA[664,35] := 251.0574;
   DATA[664,36] := 1.746067;
   DATA[664,37] := 189.743;
   DATA[664,38] := 0.000128152;
   DATA[664,39] := 1.0;
   DATA[665,0] := 2.620824;
   DATA[665,1] := 537.2917;
   DATA[665,2] := 2.0;
   DATA[665,3] := 2.0;
   DATA[665,4] := 262.1764;
   DATA[665,5] := 8.395155;
   DATA[665,6] := 327.7621;
   DATA[665,7] := 2.445007;
   DATA[665,8] := 2.0;
   DATA[665,9] := 2.0;
   DATA[665,10] := 2.0;
   DATA[665,11] := 19.70357;
   DATA[665,12] := 2.209909;
   DATA[665,13] := 988.088;
   DATA[665,14] := 1.0;
   DATA[665,15] := 2.0;
   DATA[665,16] := 1.0;
   DATA[665,17] := 1.0;
   DATA[665,18] := 1.0;
   DATA[665,19] := 2.0;
   DATA[665,20] := 148.808;
   DATA[665,21] := 155.5242;
   DATA[665,22] := 1.719027;
   DATA[665,23] := 995.937;
   DATA[665,24] := 2.0;
   DATA[665,25] := 2.0;
   DATA[665,26] := 7.878942;
   DATA[665,27] := 144.9628;
   DATA[665,28] := 263.2979;
   DATA[665,29] := 12.07383;
   DATA[665,30] := 1.73212;
   DATA[665,31] := 1.255796;
   DATA[665,32] := 0.7357808;
   DATA[665,33] := 0.3066329;
   DATA[665,34] := 2.0;
   DATA[665,35] := 251.0574;
   DATA[665,36] := 1.601897;
   DATA[665,37] := 189.743;
   DATA[665,38] := 0.000128152;
   DATA[665,39] := 1.0;
   DATA[666,0] := 2.613778;
   DATA[666,1] := 536.6245;
   DATA[666,2] := 2.0;
   DATA[666,3] := 2.0;
   DATA[666,4] := 262.1764;
   DATA[666,5] := 8.395155;
   DATA[666,6] := 327.7621;
   DATA[666,7] := 2.445007;
   DATA[666,8] := 2.0;
   DATA[666,9] := 2.0;
   DATA[666,10] := 2.0;
   DATA[666,11] := 19.70357;
   DATA[666,12] := 2.209909;
   DATA[666,13] := 987.9678;
   DATA[666,14] := 1.0;
   DATA[666,15] := 2.0;
   DATA[666,16] := 1.0;
   DATA[666,17] := 1.0;
   DATA[666,18] := 1.0;
   DATA[666,19] := 2.0;
   DATA[666,20] := 148.808;
   DATA[666,21] := 155.5242;
   DATA[666,22] := 1.718643;
   DATA[666,23] := 996.0139;
   DATA[666,24] := 2.0;
   DATA[666,25] := 2.0;
   DATA[666,26] := 7.878942;
   DATA[666,27] := 144.9628;
   DATA[666,28] := 263.2658;
   DATA[666,29] := 12.07383;
   DATA[666,30] := 1.73212;
   DATA[666,31] := 1.261432;
   DATA[666,32] := 0.7357808;
   DATA[666,33] := 0.3066329;
   DATA[666,34] := 2.0;
   DATA[666,35] := 251.0574;
   DATA[666,36] := 1.601897;
   DATA[666,37] := 189.743;
   DATA[666,38] := 0.000128152;
   DATA[666,39] := 1.0;
   DATA[667,0] := 2.598725;
   DATA[667,1] := 535.8787;
   DATA[667,2] := 2.0;
   DATA[667,3] := 2.0;
   DATA[667,4] := 262.1764;
   DATA[667,5] := 8.395155;
   DATA[667,6] := 327.7621;
   DATA[667,7] := 2.445007;
   DATA[667,8] := 2.0;
   DATA[667,9] := 2.0;
   DATA[667,10] := 2.0;
   DATA[667,11] := 19.75799;
   DATA[667,12] := 2.211575;
   DATA[667,13] := 988.0079;
   DATA[667,14] := 1.0;
   DATA[667,15] := 2.0;
   DATA[667,16] := 1.0;
   DATA[667,17] := 1.0;
   DATA[667,18] := 1.0;
   DATA[667,19] := 2.0;
   DATA[667,20] := 148.808;
   DATA[667,21] := 155.5242;
   DATA[667,22] := 1.718643;
   DATA[667,23] := 996.2446;
   DATA[667,24] := 2.0;
   DATA[667,25] := 2.0;
   DATA[667,26] := 7.878942;
   DATA[667,27] := 144.9628;
   DATA[667,28] := 263.2658;
   DATA[667,29] := 12.07383;
   DATA[667,30] := 1.729557;
   DATA[667,31] := 1.270783;
   DATA[667,32] := 0.7357808;
   DATA[667,33] := 0.3066329;
   DATA[667,34] := 2.0;
   DATA[667,35] := 251.0574;
   DATA[667,36] := 1.601897;
   DATA[667,37] := 189.743;
   DATA[667,38] := 0.000128152;
   DATA[667,39] := 1.0;
   DATA[668,0] := 2.58111;
   DATA[668,1] := 535.2899;
   DATA[668,2] := 2.0;
   DATA[668,3] := 2.0;
   DATA[668,4] := 262.1764;
   DATA[668,5] := 8.395155;
   DATA[668,6] := 327.7621;
   DATA[668,7] := 2.443341;
   DATA[668,8] := 2.0;
   DATA[668,9] := 2.0;
   DATA[668,10] := 2.0;
   DATA[668,11] := 19.77079;
   DATA[668,12] := 2.212856;
   DATA[668,13] := 987.8076;
   DATA[668,14] := 1.0;
   DATA[668,15] := 2.0;
   DATA[668,16] := 1.0;
   DATA[668,17] := 1.0;
   DATA[668,18] := 1.0;
   DATA[668,19] := 2.0;
   DATA[668,20] := 148.808;
   DATA[668,21] := 155.5242;
   DATA[668,22] := 1.718643;
   DATA[668,23] := 996.2061;
   DATA[668,24] := 2.0;
   DATA[668,25] := 2.0;
   DATA[668,26] := 7.878942;
   DATA[668,27] := 144.9628;
   DATA[668,28] := 263.2658;
   DATA[668,29] := 12.07383;
   DATA[668,30] := 1.729557;
   DATA[668,31] := 1.288843;
   DATA[668,32] := 0.7357808;
   DATA[668,33] := 0.3066329;
   DATA[668,34] := 2.0;
   DATA[668,35] := 250.9933;
   DATA[668,36] := 1.665972;
   DATA[668,37] := 189.743;
   DATA[668,38] := 0.000128152;
   DATA[668,39] := 1.0;
   DATA[669,0] := 2.564135;
   DATA[669,1] := 534.701;
   DATA[669,2] := 2.0;
   DATA[669,3] := 2.0;
   DATA[669,4] := 262.1764;
   DATA[669,5] := 8.395155;
   DATA[669,6] := 327.7621;
   DATA[669,7] := 2.443341;
   DATA[669,8] := 2.0;
   DATA[669,9] := 2.0;
   DATA[669,10] := 2.0;
   DATA[669,11] := 19.77079;
   DATA[669,12] := 2.212856;
   DATA[669,13] := 987.4071;
   DATA[669,14] := 1.0;
   DATA[669,15] := 2.0;
   DATA[669,16] := 1.0;
   DATA[669,17] := 1.0;
   DATA[669,18] := 1.0;
   DATA[669,19] := 2.0;
   DATA[669,20] := 148.808;
   DATA[669,21] := 155.5242;
   DATA[669,22] := 1.718643;
   DATA[669,23] := 995.9754;
   DATA[669,24] := 2.0;
   DATA[669,25] := 2.0;
   DATA[669,26] := 7.878942;
   DATA[669,27] := 144.9628;
   DATA[669,28] := 263.2658;
   DATA[669,29] := 12.07383;
   DATA[669,30] := 1.729557;
   DATA[669,31] := 1.300756;
   DATA[669,32] := 0.7357808;
   DATA[669,33] := 0.3066329;
   DATA[669,34] := 2.0;
   DATA[669,35] := 250.8331;
   DATA[669,36] := 1.665972;
   DATA[669,37] := 189.5988;
   DATA[669,38] := 0.000128152;
   DATA[669,39] := 1.0;
   DATA[670,0] := 2.551324;
   DATA[670,1] := 534.2693;
   DATA[670,2] := 2.0;
   DATA[670,3] := 2.0;
   DATA[670,4] := 262.1764;
   DATA[670,5] := 8.395155;
   DATA[670,6] := 327.7621;
   DATA[670,7] := 2.440265;
   DATA[670,8] := 2.0;
   DATA[670,9] := 2.0;
   DATA[670,10] := 2.0;
   DATA[670,11] := 19.77079;
   DATA[670,12] := 2.21055;
   DATA[670,13] := 987.3671;
   DATA[670,14] := 1.0;
   DATA[670,15] := 2.0;
   DATA[670,16] := 1.0;
   DATA[670,17] := 1.0;
   DATA[670,18] := 1.0;
   DATA[670,19] := 2.0;
   DATA[670,20] := 148.808;
   DATA[670,21] := 155.5242;
   DATA[670,22] := 1.718643;
   DATA[670,23] := 996.1292;
   DATA[670,24] := 2.0;
   DATA[670,25] := 2.0;
   DATA[670,26] := 7.878942;
   DATA[670,27] := 144.9628;
   DATA[670,28] := 263.2658;
   DATA[670,29] := 12.07383;
   DATA[670,30] := 1.730454;
   DATA[670,31] := 1.301524;
   DATA[670,32] := 0.7357808;
   DATA[670,33] := 0.3066329;
   DATA[670,34] := 2.0;
   DATA[670,35] := 250.8331;
   DATA[670,36] := 1.665972;
   DATA[670,37] := 189.5988;
   DATA[670,38] := 0.000128152;
   DATA[670,39] := 1.0;
   DATA[671,0] := 2.532748;
   DATA[671,1] := 533.8375;
   DATA[671,2] := 2.0;
   DATA[671,3] := 2.0;
   DATA[671,4] := 262.1764;
   DATA[671,5] := 8.395155;
   DATA[671,6] := 327.7621;
   DATA[671,7] := 2.439753;
   DATA[671,8] := 2.0;
   DATA[671,9] := 2.0;
   DATA[671,10] := 2.0;
   DATA[671,11] := 19.77079;
   DATA[671,12] := 2.21055;
   DATA[671,13] := 987.6074;
   DATA[671,14] := 1.0;
   DATA[671,15] := 2.0;
   DATA[671,16] := 1.0;
   DATA[671,17] := 1.0;
   DATA[671,18] := 1.0;
   DATA[671,19] := 2.0;
   DATA[671,20] := 148.808;
   DATA[671,21] := 155.5242;
   DATA[671,22] := 1.718643;
   DATA[671,23] := 996.0523;
   DATA[671,24] := 2.0;
   DATA[671,25] := 2.0;
   DATA[671,26] := 7.878942;
   DATA[671,27] := 144.9628;
   DATA[671,28] := 263.1377;
   DATA[671,29] := 12.07383;
   DATA[671,30] := 1.731351;
   DATA[671,31] := 1.296401;
   DATA[671,32] := 0.7357808;
   DATA[671,33] := 0.3080421;
   DATA[671,34] := 2.0;
   DATA[671,35] := 250.9773;
   DATA[671,36] := 1.665972;
   DATA[671,37] := 189.6789;
   DATA[671,38] := 0.000128152;
   DATA[671,39] := 1.0;
   DATA[672,0] := 2.519297;
   DATA[672,1] := 534.3478;
   DATA[672,2] := 2.0;
   DATA[672,3] := 2.0;
   DATA[672,4] := 262.1764;
   DATA[672,5] := 8.395155;
   DATA[672,6] := 327.7621;
   DATA[672,7] := 2.439753;
   DATA[672,8] := 2.0;
   DATA[672,9] := 2.0;
   DATA[672,10] := 2.0;
   DATA[672,11] := 19.71637;
   DATA[672,12] := 2.21055;
   DATA[672,13] := 987.7676;
   DATA[672,14] := 1.0;
   DATA[672,15] := 2.0;
   DATA[672,16] := 1.0;
   DATA[672,17] := 1.0;
   DATA[672,18] := 1.0;
   DATA[672,19] := 2.0;
   DATA[672,20] := 148.808;
   DATA[672,21] := 155.5242;
   DATA[672,22] := 1.718643;
   DATA[672,23] := 996.1292;
   DATA[672,24] := 2.0;
   DATA[672,25] := 2.0;
   DATA[672,26] := 7.878942;
   DATA[672,27] := 144.8603;
   DATA[672,28] := 263.1377;
   DATA[672,29] := 12.07383;
   DATA[672,30] := 1.731351;
   DATA[672,31] := 1.282183;
   DATA[672,32] := 0.7357808;
   DATA[672,33] := 0.3084905;
   DATA[672,34] := 2.0;
   DATA[672,35] := 250.9773;
   DATA[672,36] := 1.778105;
   DATA[672,37] := 189.8391;
   DATA[672,38] := 0.000128152;
   DATA[672,39] := 1.0;
   DATA[673,0] := 2.498799;
   DATA[673,1] := 534.8581;
   DATA[673,2] := 2.0;
   DATA[673,3] := 2.0;
   DATA[673,4] := 262.1764;
   DATA[673,5] := 8.395155;
   DATA[673,6] := 327.7621;
   DATA[673,7] := 2.439753;
   DATA[673,8] := 2.0;
   DATA[673,9] := 2.0;
   DATA[673,10] := 2.0;
   DATA[673,11] := 19.71637;
   DATA[673,12] := 2.209525;
   DATA[673,13] := 988.0079;
   DATA[673,14] := 1.0;
   DATA[673,15] := 2.0;
   DATA[673,16] := 1.0;
   DATA[673,17] := 1.0;
   DATA[673,18] := 1.0;
   DATA[673,19] := 2.0;
   DATA[673,20] := 148.808;
   DATA[673,21] := 155.5242;
   DATA[673,22] := 1.720565;
   DATA[673,23] := 996.3215;
   DATA[673,24] := 2.0;
   DATA[673,25] := 2.0;
   DATA[673,26] := 7.878942;
   DATA[673,27] := 144.8603;
   DATA[673,28] := 263.1377;
   DATA[673,29] := 12.07383;
   DATA[673,30] := 1.729172;
   DATA[673,31] := 1.28436;
   DATA[673,32] := 0.7352687;
   DATA[673,33] := 0.3084905;
   DATA[673,34] := 2.0;
   DATA[673,35] := 251.1535;
   DATA[673,36] := 1.778105;
   DATA[673,37] := 189.8391;
   DATA[673,38] := 0.000128152;
   DATA[673,39] := 1.0;
   DATA[674,0] := 2.486308;
   DATA[674,1] := 535.2114;
   DATA[674,2] := 2.0;
   DATA[674,3] := 2.0;
   DATA[674,4] := 262.1764;
   DATA[674,5] := 8.395155;
   DATA[674,6] := 327.7621;
   DATA[674,7] := 2.441803;
   DATA[674,8] := 2.0;
   DATA[674,9] := 2.0;
   DATA[674,10] := 2.0;
   DATA[674,11] := 19.71637;
   DATA[674,12] := 2.209397;
   DATA[674,13] := 988.4084;
   DATA[674,14] := 1.0;
   DATA[674,15] := 2.0;
   DATA[674,16] := 1.0;
   DATA[674,17] := 1.0;
   DATA[674,18] := 1.0;
   DATA[674,19] := 2.0;
   DATA[674,20] := 148.808;
   DATA[674,21] := 155.5242;
   DATA[674,22] := 1.72159;
   DATA[674,23] := 996.5137;
   DATA[674,24] := 2.0;
   DATA[674,25] := 2.0;
   DATA[674,26] := 7.878942;
   DATA[674,27] := 144.7065;
   DATA[674,28] := 263.1377;
   DATA[674,29] := 12.07383;
   DATA[674,30] := 1.729172;
   DATA[674,31] := 1.290637;
   DATA[674,32] := 0.7352687;
   DATA[674,33] := 0.3069532;
   DATA[674,34] := 2.0;
   DATA[674,35] := 251.1535;
   DATA[674,36] := 1.778105;
   DATA[674,37] := 189.8391;
   DATA[674,38] := 0.000128152;
   DATA[674,39] := 1.0;
   DATA[675,0] := 2.474778;
   DATA[675,1] := 535.9964;
   DATA[675,2] := 2.0;
   DATA[675,3] := 2.0;
   DATA[675,4] := 262.1764;
   DATA[675,5] := 8.395155;
   DATA[675,6] := 327.7108;
   DATA[675,7] := 2.441803;
   DATA[675,8] := 2.0;
   DATA[675,9] := 2.0;
   DATA[675,10] := 2.0;
   DATA[675,11] := 19.71637;
   DATA[675,12] := 2.209397;
   DATA[675,13] := 988.6487;
   DATA[675,14] := 1.0;
   DATA[675,15] := 2.0;
   DATA[675,16] := 1.0;
   DATA[675,17] := 1.0;
   DATA[675,18] := 1.0;
   DATA[675,19] := 2.0;
   DATA[675,20] := 148.808;
   DATA[675,21] := 155.5242;
   DATA[675,22] := 1.72159;
   DATA[675,23] := 996.3984;
   DATA[675,24] := 2.0;
   DATA[675,25] := 2.0;
   DATA[675,26] := 7.878942;
   DATA[675,27] := 144.7065;
   DATA[675,28] := 263.1377;
   DATA[675,29] := 12.07383;
   DATA[675,30] := 1.729172;
   DATA[675,31] := 1.291149;
   DATA[675,32] := 0.7352687;
   DATA[675,33] := 0.3069532;
   DATA[675,34] := 2.0;
   DATA[675,35] := 251.1535;
   DATA[675,36] := 1.778105;
   DATA[675,37] := 189.8391;
   DATA[675,38] := 0.000128152;
   DATA[675,39] := 1.0;
   DATA[676,0] := 2.458444;
   DATA[676,1] := 536.6245;
   DATA[676,2] := 2.0;
   DATA[676,3] := 2.0;
   DATA[676,4] := 262.1764;
   DATA[676,5] := 8.395155;
   DATA[676,6] := 327.6083;
   DATA[676,7] := 2.440521;
   DATA[676,8] := 2.0;
   DATA[676,9] := 2.0;
   DATA[676,10] := 2.0;
   DATA[676,11] := 19.77079;
   DATA[676,12] := 2.209397;
   DATA[676,13] := 988.6888;
   DATA[676,14] := 1.0;
   DATA[676,15] := 2.0;
   DATA[676,16] := 1.0;
   DATA[676,17] := 1.0;
   DATA[676,18] := 1.0;
   DATA[676,19] := 2.0;
   DATA[676,20] := 148.808;
   DATA[676,21] := 155.5242;
   DATA[676,22] := 1.719924;
   DATA[676,23] := 996.8214;
   DATA[676,24] := 2.0;
   DATA[676,25] := 2.0;
   DATA[676,26] := 7.878942;
   DATA[676,27] := 144.7065;
   DATA[676,28] := 263.1377;
   DATA[676,29] := 12.07383;
   DATA[676,30] := 1.729172;
   DATA[676,31] := 1.292046;
   DATA[676,32] := 0.7352687;
   DATA[676,33] := 0.3063127;
   DATA[676,34] := 2.0;
   DATA[676,35] := 251.2657;
   DATA[676,36] := 1.778105;
   DATA[676,37] := 189.9353;
   DATA[676,38] := 0.000128152;
   DATA[676,39] := 1.0;
   DATA[677,0] := 2.443391;
   DATA[677,1] := 536.8992;
   DATA[677,2] := 2.0;
   DATA[677,3] := 2.0;
   DATA[677,4] := 262.1764;
   DATA[677,5] := 8.395155;
   DATA[677,6] := 327.6083;
   DATA[677,7] := 2.439881;
   DATA[677,8] := 2.0;
   DATA[677,9] := 2.0;
   DATA[677,10] := 2.0;
   DATA[677,11] := 19.77079;
   DATA[677,12] := 2.209397;
   DATA[677,13] := 988.4885;
   DATA[677,14] := 1.0;
   DATA[677,15] := 2.0;
   DATA[677,16] := 1.0;
   DATA[677,17] := 1.0;
   DATA[677,18] := 1.0;
   DATA[677,19] := 2.0;
   DATA[677,20] := 148.808;
   DATA[677,21] := 155.5242;
   DATA[677,22] := 1.719924;
   DATA[677,23] := 997.0905;
   DATA[677,24] := 2.0;
   DATA[677,25] := 2.0;
   DATA[677,26] := 7.878942;
   DATA[677,27] := 144.7065;
   DATA[677,28] := 263.1377;
   DATA[677,29] := 12.07383;
   DATA[677,30] := 1.729172;
   DATA[677,31] := 1.288587;
   DATA[677,32] := 0.7352687;
   DATA[677,33] := 0.3063127;
   DATA[677,34] := 2.0;
   DATA[677,35] := 251.2657;
   DATA[677,36] := 1.730048;
   DATA[677,37] := 189.9353;
   DATA[677,38] := 0.000128152;
   DATA[677,39] := 1.0;
   DATA[678,0] := 2.431861;
   DATA[678,1] := 537.7628;
   DATA[678,2] := 2.0;
   DATA[678,3] := 2.0;
   DATA[678,4] := 262.1764;
   DATA[678,5] := 8.396757;
   DATA[678,6] := 327.6083;
   DATA[678,7] := 2.439881;
   DATA[678,8] := 2.0;
   DATA[678,9] := 2.0;
   DATA[678,10] := 2.0;
   DATA[678,11] := 19.77079;
   DATA[678,12] := 2.209397;
   DATA[678,13] := 988.5687;
   DATA[678,14] := 1.0;
   DATA[678,15] := 2.0;
   DATA[678,16] := 1.0;
   DATA[678,17] := 1.0;
   DATA[678,18] := 1.0;
   DATA[678,19] := 2.0;
   DATA[678,20] := 148.808;
   DATA[678,21] := 155.5242;
   DATA[678,22] := 1.719924;
   DATA[678,23] := 997.475;
   DATA[678,24] := 2.0;
   DATA[678,25] := 2.0;
   DATA[678,26] := 7.878942;
   DATA[678,27] := 144.7065;
   DATA[678,28] := 263.1377;
   DATA[678,29] := 12.26609;
   DATA[678,30] := 1.729172;
   DATA[678,31] := 1.28167;
   DATA[678,32] := 0.7352687;
   DATA[678,33] := 0.3063127;
   DATA[678,34] := 2.0;
   DATA[678,35] := 251.2657;
   DATA[678,36] := 1.730048;
   DATA[678,37] := 189.9353;
   DATA[678,38] := 0.000128152;
   DATA[678,39] := 1.0;
   DATA[679,0] := 2.43058;
   DATA[679,1] := 537.6058;
   DATA[679,2] := 2.0;
   DATA[679,3] := 2.0;
   DATA[679,4] := 262.1764;
   DATA[679,5] := 8.396757;
   DATA[679,6] := 327.6083;
   DATA[679,7] := 2.439881;
   DATA[679,8] := 2.0;
   DATA[679,9] := 2.0;
   DATA[679,10] := 2.0;
   DATA[679,11] := 19.77079;
   DATA[679,12] := 2.209397;
   DATA[679,13] := 988.8491;
   DATA[679,14] := 1.0;
   DATA[679,15] := 2.0;
   DATA[679,16] := 1.0;
   DATA[679,17] := 1.0;
   DATA[679,18] := 1.0;
   DATA[679,19] := 2.0;
   DATA[679,20] := 148.808;
   DATA[679,21] := 155.5242;
   DATA[679,22] := 1.719924;
   DATA[679,23] := 997.3212;
   DATA[679,24] := 2.0;
   DATA[679,25] := 2.0;
   DATA[679,26] := 7.878942;
   DATA[679,27] := 144.7065;
   DATA[679,28] := 263.1377;
   DATA[679,29] := 12.26609;
   DATA[679,30] := 1.730582;
   DATA[679,31] := 1.28167;
   DATA[679,32] := 0.7352687;
   DATA[679,33] := 0.3063127;
   DATA[679,34] := 2.0;
   DATA[679,35] := 251.2657;
   DATA[679,36] := 1.730048;
   DATA[679,37] := 189.9353;
   DATA[679,38] := 0.000128152;
   DATA[679,39] := 1.0;
   DATA[680,0] := 2.43058;
   DATA[680,1] := 537.5665;
   DATA[680,2] := 2.0;
   DATA[680,3] := 2.0;
   DATA[680,4] := 262.1764;
   DATA[680,5] := 8.396757;
   DATA[680,6] := 327.6083;
   DATA[680,7] := 2.439881;
   DATA[680,8] := 2.0;
   DATA[680,9] := 2.0;
   DATA[680,10] := 2.0;
   DATA[680,11] := 19.77079;
   DATA[680,12] := 2.209397;
   DATA[680,13] := 989.0093;
   DATA[680,14] := 1.0;
   DATA[680,15] := 2.0;
   DATA[680,16] := 1.0;
   DATA[680,17] := 1.0;
   DATA[680,18] := 1.0;
   DATA[680,19] := 2.0;
   DATA[680,20] := 148.808;
   DATA[680,21] := 155.5242;
   DATA[680,22] := 1.719924;
   DATA[680,23] := 997.7441;
   DATA[680,24] := 2.0;
   DATA[680,25] := 2.0;
   DATA[680,26] := 7.878942;
   DATA[680,27] := 144.7065;
   DATA[680,28] := 263.1377;
   DATA[680,29] := 12.26609;
   DATA[680,30] := 1.731095;
   DATA[680,31] := 1.272192;
   DATA[680,32] := 0.7352687;
   DATA[680,33] := 0.305608;
   DATA[680,34] := 2.0;
   DATA[680,35] := 251.2657;
   DATA[680,36] := 1.730048;
   DATA[680,37] := 189.9353;
   DATA[680,38] := 0.000128152;
   DATA[680,39] := 1.0;
   DATA[681,0] := 2.456843;
   DATA[681,1] := 537.6843;
   DATA[681,2] := 2.0;
   DATA[681,3] := 2.0;
   DATA[681,4] := 262.1764;
   DATA[681,5] := 8.396757;
   DATA[681,6] := 327.6083;
   DATA[681,7] := 2.439881;
   DATA[681,8] := 2.0;
   DATA[681,9] := 2.0;
   DATA[681,10] := 2.0;
   DATA[681,11] := 19.76759;
   DATA[681,12] := 2.209397;
   DATA[681,13] := 988.6087;
   DATA[681,14] := 1.0;
   DATA[681,15] := 2.0;
   DATA[681,16] := 1.0;
   DATA[681,17] := 1.0;
   DATA[681,18] := 1.0;
   DATA[681,19] := 2.0;
   DATA[681,20] := 148.808;
   DATA[681,21] := 155.5242;
   DATA[681,22] := 1.719924;
   DATA[681,23] := 998.1671;
   DATA[681,24] := 2.0;
   DATA[681,25] := 2.0;
   DATA[681,26] := 7.878942;
   DATA[681,27] := 144.7065;
   DATA[681,28] := 263.1377;
   DATA[681,29] := 12.03538;
   DATA[681,30] := 1.731095;
   DATA[681,31] := 1.272192;
   DATA[681,32] := 0.7352687;
   DATA[681,33] := 0.3058002;
   DATA[681,34] := 2.0;
   DATA[681,35] := 251.2657;
   DATA[681,36] := 1.730048;
   DATA[681,37] := 189.9353;
   DATA[681,38] := 0.000128152;
   DATA[681,39] := 1.0;
   DATA[682,0] := 2.502642;
   DATA[682,1] := 537.8806;
   DATA[682,2] := 2.0;
   DATA[682,3] := 2.0;
   DATA[682,4] := 262.1764;
   DATA[682,5] := 8.396757;
   DATA[682,6] := 327.7108;
   DATA[682,7] := 2.439881;
   DATA[682,8] := 2.0;
   DATA[682,9] := 2.0;
   DATA[682,10] := 2.0;
   DATA[682,11] := 19.73558;
   DATA[682,12] := 2.211575;
   DATA[682,13] := 988.9692;
   DATA[682,14] := 1.0;
   DATA[682,15] := 2.0;
   DATA[682,16] := 1.0;
   DATA[682,17] := 1.0;
   DATA[682,18] := 1.0;
   DATA[682,19] := 2.0;
   DATA[682,20] := 148.808;
   DATA[682,21] := 155.7806;
   DATA[682,22] := 1.719924;
   DATA[682,23] := 998.0902;
   DATA[682,24] := 2.0;
   DATA[682,25] := 2.0;
   DATA[682,26] := 7.878942;
   DATA[682,27] := 144.7065;
   DATA[682,28] := 263.1377;
   DATA[682,29] := 11.92002;
   DATA[682,30] := 1.731095;
   DATA[682,31] := 1.279237;
   DATA[682,32] := 0.7352687;
   DATA[682,33] := 0.3068251;
   DATA[682,34] := 2.0;
   DATA[682,35] := 251.2657;
   DATA[682,36] := 1.730048;
   DATA[682,37] := 189.9353;
   DATA[682,38] := 0.000128152;
   DATA[682,39] := 1.0;
   DATA[683,0] := 2.542677;
   DATA[683,1] := 537.645;
   DATA[683,2] := 2.0;
   DATA[683,3] := 2.0;
   DATA[683,4] := 262.1764;
   DATA[683,5] := 8.396757;
   DATA[683,6] := 327.7108;
   DATA[683,7] := 2.439881;
   DATA[683,8] := 2.0;
   DATA[683,9] := 2.0;
   DATA[683,10] := 2.0;
   DATA[683,11] := 19.73558;
   DATA[683,12] := 2.212984;
   DATA[683,13] := 989.4899;
   DATA[683,14] := 1.0;
   DATA[683,15] := 2.0;
   DATA[683,16] := 1.0;
   DATA[683,17] := 1.0;
   DATA[683,18] := 1.0;
   DATA[683,19] := 2.0;
   DATA[683,20] := 148.808;
   DATA[683,21] := 155.7806;
   DATA[683,22] := 1.719924;
   DATA[683,23] := 998.3209;
   DATA[683,24] := 2.0;
   DATA[683,25] := 2.0;
   DATA[683,26] := 7.878942;
   DATA[683,27] := 144.7065;
   DATA[683,28] := 263.1377;
   DATA[683,29] := 11.92002;
   DATA[683,30] := 1.731095;
   DATA[683,31] := 1.297041;
   DATA[683,32] := 0.7352687;
   DATA[683,33] := 0.3068251;
   DATA[683,34] := 2.0;
   DATA[683,35] := 251.2657;
   DATA[683,36] := 1.730048;
   DATA[683,37] := 189.9353;
   DATA[683,38] := 0.000128152;
   DATA[683,39] := 1.0;
   DATA[684,0] := 2.575345;
   DATA[684,1] := 537.4488;
   DATA[684,2] := 2.0;
   DATA[684,3] := 2.0;
   DATA[684,4] := 262.1764;
   DATA[684,5] := 8.396757;
   DATA[684,6] := 327.7108;
   DATA[684,7] := 2.441675;
   DATA[684,8] := 2.0;
   DATA[684,9] := 2.0;
   DATA[684,10] := 2.0;
   DATA[684,11] := 19.70357;
   DATA[684,12] := 2.215802;
   DATA[684,13] := 989.8504;
   DATA[684,14] := 1.0;
   DATA[684,15] := 2.0;
   DATA[684,16] := 1.0;
   DATA[684,17] := 1.0;
   DATA[684,18] := 1.0;
   DATA[684,19] := 2.0;
   DATA[684,20] := 148.808;
   DATA[684,21] := 155.7806;
   DATA[684,22] := 1.719924;
   DATA[684,23] := 998.4363;
   DATA[684,24] := 2.0;
   DATA[684,25] := 2.0;
   DATA[684,26] := 7.878942;
   DATA[684,27] := 144.7065;
   DATA[684,28] := 263.1377;
   DATA[684,29] := 11.92002;
   DATA[684,30] := 1.731095;
   DATA[684,31] := 1.311643;
   DATA[684,32] := 0.7352687;
   DATA[684,33] := 0.3068251;
   DATA[684,34] := 2.0;
   DATA[684,35] := 251.2657;
   DATA[684,36] := 1.810143;
   DATA[684,37] := 190.0955;
   DATA[684,38] := 0.000128152;
   DATA[684,39] := 1.0;
   DATA[685,0] := 2.612497;
   DATA[685,1] := 537.0955;
   DATA[685,2] := 2.0;
   DATA[685,3] := 2.0;
   DATA[685,4] := 262.1764;
   DATA[685,5] := 8.396437;
   DATA[685,6] := 327.7108;
   DATA[685,7] := 2.4427;
   DATA[685,8] := 2.0;
   DATA[685,9] := 2.0;
   DATA[685,10] := 2.0;
   DATA[685,11] := 19.70357;
   DATA[685,12] := 2.215802;
   DATA[685,13] := 989.7703;
   DATA[685,14] := 1.0;
   DATA[685,15] := 2.0;
   DATA[685,16] := 1.0;
   DATA[685,17] := 1.0;
   DATA[685,18] := 1.0;
   DATA[685,19] := 2.0;
   DATA[685,20] := 148.808;
   DATA[685,21] := 155.7806;
   DATA[685,22] := 1.721847;
   DATA[685,23] := 998.5516;
   DATA[685,24] := 2.0;
   DATA[685,25] := 2.0;
   DATA[685,26] := 7.878942;
   DATA[685,27] := 144.7065;
   DATA[685,28] := 263.1377;
   DATA[685,29] := 11.92002;
   DATA[685,30] := 1.731095;
   DATA[685,31] := 1.305879;
   DATA[685,32] := 0.7352687;
   DATA[685,33] := 0.3068251;
   DATA[685,34] := 2.0;
   DATA[685,35] := 251.458;
   DATA[685,36] := 1.810143;
   DATA[685,37] := 190.0955;
   DATA[685,38] := 0.000128152;
   DATA[685,39] := 1.0;
   DATA[686,0] := 2.635237;
   DATA[686,1] := 537.017;
   DATA[686,2] := 2.0;
   DATA[686,3] := 2.0;
   DATA[686,4] := 262.1764;
   DATA[686,5] := 8.396437;
   DATA[686,6] := 327.7108;
   DATA[686,7] := 2.442956;
   DATA[686,8] := 2.0;
   DATA[686,9] := 2.0;
   DATA[686,10] := 2.0;
   DATA[686,11] := 19.70357;
   DATA[686,12] := 2.214906;
   DATA[686,13] := 989.8904;
   DATA[686,14] := 1.0;
   DATA[686,15] := 2.0;
   DATA[686,16] := 1.0;
   DATA[686,17] := 1.0;
   DATA[686,18] := 1.0;
   DATA[686,19] := 2.0;
   DATA[686,20] := 148.808;
   DATA[686,21] := 155.7806;
   DATA[686,22] := 1.721847;
   DATA[686,23] := 998.8208;
   DATA[686,24] := 2.0;
   DATA[686,25] := 2.0;
   DATA[686,26] := 7.878942;
   DATA[686,27] := 144.7065;
   DATA[686,28] := 263.1377;
   DATA[686,29] := 11.92002;
   DATA[686,30] := 1.731095;
   DATA[686,31] := 1.300372;
   DATA[686,32] := 0.7352687;
   DATA[686,33] := 0.3068251;
   DATA[686,34] := 2.0;
   DATA[686,35] := 251.506;
   DATA[686,36] := 1.810143;
   DATA[686,37] := 190.0955;
   DATA[686,38] := 0.000128152;
   DATA[686,39] := 1.0;
   DATA[687,0] := 2.655414;
   DATA[687,1] := 536.3889;
   DATA[687,2] := 2.0;
   DATA[687,3] := 2.0;
   DATA[687,4] := 262.1764;
   DATA[687,5] := 8.396437;
   DATA[687,6] := 327.7108;
   DATA[687,7] := 2.440906;
   DATA[687,8] := 2.0;
   DATA[687,9] := 2.0;
   DATA[687,10] := 2.0;
   DATA[687,11] := 19.70357;
   DATA[687,12] := 2.214906;
   DATA[687,13] := 989.8103;
   DATA[687,14] := 1.0;
   DATA[687,15] := 2.0;
   DATA[687,16] := 1.0;
   DATA[687,17] := 1.0;
   DATA[687,18] := 1.0;
   DATA[687,19] := 2.0;
   DATA[687,20] := 148.808;
   DATA[687,21] := 155.7806;
   DATA[687,22] := 1.721847;
   DATA[687,23] := 998.9362;
   DATA[687,24] := 2.0;
   DATA[687,25] := 2.0;
   DATA[687,26] := 7.878942;
   DATA[687,27] := 144.7065;
   DATA[687,28] := 263.1377;
   DATA[687,29] := 11.92002;
   DATA[687,30] := 1.731095;
   DATA[687,31] := 1.283464;
   DATA[687,32] := 0.7352687;
   DATA[687,33] := 0.3068251;
   DATA[687,34] := 2.0;
   DATA[687,35] := 251.506;
   DATA[687,36] := 1.810143;
   DATA[687,37] := 190.0955;
   DATA[687,38] := 0.000128152;
   DATA[687,39] := 1.0;
   DATA[688,0] := 2.657016;
   DATA[688,1] := 536.86;
   DATA[688,2] := 2.0;
   DATA[688,3] := 2.0;
   DATA[688,4] := 262.1764;
   DATA[688,5] := 8.396437;
   DATA[688,6] := 327.7108;
   DATA[688,7] := 2.439881;
   DATA[688,8] := 2.0;
   DATA[688,9] := 2.0;
   DATA[688,10] := 2.0;
   DATA[688,11] := 19.70357;
   DATA[688,12] := 2.214906;
   DATA[688,13] := 989.7703;
   DATA[688,14] := 1.0;
   DATA[688,15] := 2.0;
   DATA[688,16] := 1.0;
   DATA[688,17] := 1.0;
   DATA[688,18] := 1.0;
   DATA[688,19] := 2.0;
   DATA[688,20] := 148.808;
   DATA[688,21] := 155.7806;
   DATA[688,22] := 1.720309;
   DATA[688,23] := 999.2438;
   DATA[688,24] := 2.0;
   DATA[688,25] := 2.0;
   DATA[688,26] := 7.878942;
   DATA[688,27] := 144.7065;
   DATA[688,28] := 263.1377;
   DATA[688,29] := 11.92002;
   DATA[688,30] := 1.731095;
   DATA[688,31] := 1.271935;
   DATA[688,32] := 0.7352687;
   DATA[688,33] := 0.3068251;
   DATA[688,34] := 2.0;
   DATA[688,35] := 251.2657;
   DATA[688,36] := 1.810143;
   DATA[688,37] := 190.0795;
   DATA[688,38] := 0.000128152;
   DATA[688,39] := 1.0;
   DATA[689,0] := 2.657016;
   DATA[689,1] := 536.86;
   DATA[689,2] := 2.0;
   DATA[689,3] := 2.0;
   DATA[689,4] := 262.1764;
   DATA[689,5] := 8.396437;
   DATA[689,6] := 327.7108;
   DATA[689,7] := 2.439881;
   DATA[689,8] := 2.0;
   DATA[689,9] := 2.0;
   DATA[689,10] := 2.0;
   DATA[689,11] := 19.70357;
   DATA[689,12] := 2.214906;
   DATA[689,13] := 989.7703;
   DATA[689,14] := 1.0;
   DATA[689,15] := 2.0;
   DATA[689,16] := 1.0;
   DATA[689,17] := 1.0;
   DATA[689,18] := 1.0;
   DATA[689,19] := 2.0;
   DATA[689,20] := 148.808;
   DATA[689,21] := 155.7806;
   DATA[689,22] := 1.720309;
   DATA[689,23] := 999.2438;
   DATA[689,24] := 2.0;
   DATA[689,25] := 2.0;
   DATA[689,26] := 7.878942;
   DATA[689,27] := 144.7065;
   DATA[689,28] := 263.1377;
   DATA[689,29] := 11.92002;
   DATA[689,30] := 1.731095;
   DATA[689,31] := 1.271935;
   DATA[689,32] := 0.7352687;
   DATA[689,33] := 0.3068251;
   DATA[689,34] := 2.0;
   DATA[689,35] := 251.2657;
   DATA[689,36] := 1.810143;
   DATA[689,37] := 190.0795;
   DATA[689,38] := 0.000128152;
   DATA[689,39] := 1.0;
   DATA[690,0] := 2.645165;
   DATA[690,1] := 537.0955;
   DATA[690,2] := 2.0;
   DATA[690,3] := 2.0;
   DATA[690,4] := 262.1764;
   DATA[690,5] := 8.395475;
   DATA[690,6] := 327.7108;
   DATA[690,7] := 2.439881;
   DATA[690,8] := 2.0;
   DATA[690,9] := 2.0;
   DATA[690,10] := 2.0;
   DATA[690,11] := 19.70357;
   DATA[690,12] := 2.214906;
   DATA[690,13] := 989.7703;
   DATA[690,14] := 1.0;
   DATA[690,15] := 2.0;
   DATA[690,16] := 1.0;
   DATA[690,17] := 1.0;
   DATA[690,18] := 1.0;
   DATA[690,19] := 2.0;
   DATA[690,20] := 148.808;
   DATA[690,21] := 155.7806;
   DATA[690,22] := 1.720309;
   DATA[690,23] := 999.2053;
   DATA[690,24] := 2.0;
   DATA[690,25] := 2.0;
   DATA[690,26] := 7.878942;
   DATA[690,27] := 144.7065;
   DATA[690,28] := 263.1377;
   DATA[690,29] := 11.92002;
   DATA[690,30] := 1.731095;
   DATA[690,31] := 1.268349;
   DATA[690,32] := 0.7352687;
   DATA[690,33] := 0.3068251;
   DATA[690,34] := 2.0;
   DATA[690,35] := 251.2657;
   DATA[690,36] := 1.69801;
   DATA[690,37] := 189.9193;
   DATA[690,38] := 0.000128152;
   DATA[690,39] := 1.0;
   DATA[691,0] := 2.62755;
   DATA[691,1] := 537.488;
   DATA[691,2] := 2.0;
   DATA[691,3] := 2.0;
   DATA[691,4] := 262.1764;
   DATA[691,5] := 8.395475;
   DATA[691,6] := 327.7108;
   DATA[691,7] := 2.439881;
   DATA[691,8] := 2.0;
   DATA[691,9] := 2.0;
   DATA[691,10] := 2.0;
   DATA[691,11] := 19.73558;
   DATA[691,12] := 2.214906;
   DATA[691,13] := 989.4498;
   DATA[691,14] := 1.0;
   DATA[691,15] := 2.0;
   DATA[691,16] := 1.0;
   DATA[691,17] := 1.0;
   DATA[691,18] := 1.0;
   DATA[691,19] := 2.0;
   DATA[691,20] := 148.808;
   DATA[691,21] := 155.7037;
   DATA[691,22] := 1.720309;
   DATA[691,23] := 998.8208;
   DATA[691,24] := 2.0;
   DATA[691,25] := 2.0;
   DATA[691,26] := 7.878942;
   DATA[691,27] := 144.7065;
   DATA[691,28] := 263.1377;
   DATA[691,29] := 11.95847;
   DATA[691,30] := 1.73071;
   DATA[691,31] := 1.262329;
   DATA[691,32] := 0.7352687;
   DATA[691,33] := 0.3064407;
   DATA[691,34] := 2.0;
   DATA[691,35] := 251.2657;
   DATA[691,36] := 1.69801;
   DATA[691,37] := 189.9193;
   DATA[691,38] := 0.000128152;
   DATA[691,39] := 1.0;
   DATA[692,0] := 2.622105;
   DATA[692,1] := 537.5665;
   DATA[692,2] := 2.0;
   DATA[692,3] := 2.0;
   DATA[692,4] := 262.1764;
   DATA[692,5] := 8.395475;
   DATA[692,6] := 327.7108;
   DATA[692,7] := 2.439881;
   DATA[692,8] := 2.0;
   DATA[692,9] := 2.0;
   DATA[692,10] := 2.0;
   DATA[692,11] := 19.73878;
   DATA[692,12] := 2.212984;
   DATA[692,13] := 989.4899;
   DATA[692,14] := 1.0;
   DATA[692,15] := 2.0;
   DATA[692,16] := 1.0;
   DATA[692,17] := 1.0;
   DATA[692,18] := 1.0;
   DATA[692,19] := 2.0;
   DATA[692,20] := 148.808;
   DATA[692,21] := 155.5499;
   DATA[692,22] := 1.720309;
   DATA[692,23] := 999.0131;
   DATA[692,24] := 2.0;
   DATA[692,25] := 2.0;
   DATA[692,26] := 7.878942;
   DATA[692,27] := 144.7321;
   DATA[692,28] := 263.1377;
   DATA[692,29] := 12.11228;
   DATA[692,30] := 1.7293;
   DATA[692,31] := 1.270014;
   DATA[692,32] := 0.7352687;
   DATA[692,33] := 0.3064407;
   DATA[692,34] := 2.0;
   DATA[692,35] := 251.2657;
   DATA[692,36] := 1.69801;
   DATA[692,37] := 189.9193;
   DATA[692,38] := 0.000128152;
   DATA[692,39] := 1.0;
   DATA[693,0] := 2.613778;
   DATA[693,1] := 538.0768;
   DATA[693,2] := 2.0;
   DATA[693,3] := 2.0;
   DATA[693,4] := 262.1764;
   DATA[693,5] := 8.395475;
   DATA[693,6] := 327.7108;
   DATA[693,7] := 2.439881;
   DATA[693,8] := 2.0;
   DATA[693,9] := 2.0;
   DATA[693,10] := 2.0;
   DATA[693,11] := 19.73878;
   DATA[693,12] := 2.210806;
   DATA[693,13] := 989.3698;
   DATA[693,14] := 1.0;
   DATA[693,15] := 2.0;
   DATA[693,16] := 1.0;
   DATA[693,17] := 1.0;
   DATA[693,18] := 1.0;
   DATA[693,19] := 2.0;
   DATA[693,20] := 148.808;
   DATA[693,21] := 155.5499;
   DATA[693,22] := 1.720309;
   DATA[693,23] := 998.8208;
   DATA[693,24] := 2.0;
   DATA[693,25] := 2.0;
   DATA[693,26] := 7.878942;
   DATA[693,27] := 144.7321;
   DATA[693,28] := 263.1377;
   DATA[693,29] := 12.11228;
   DATA[693,30] := 1.7293;
   DATA[693,31] := 1.281542;
   DATA[693,32] := 0.7352687;
   DATA[693,33] := 0.3064407;
   DATA[693,34] := 2.0;
   DATA[693,35] := 251.0734;
   DATA[693,36] := 1.69801;
   DATA[693,37] := 189.9193;
   DATA[693,38] := 0.000128152;
   DATA[693,39] := 1.0;
   DATA[694,0] := 2.595522;
   DATA[694,1] := 537.8413;
   DATA[694,2] := 2.0;
   DATA[694,3] := 2.0;
   DATA[694,4] := 262.1764;
   DATA[694,5] := 8.395475;
   DATA[694,6] := 327.7108;
   DATA[694,7] := 2.439881;
   DATA[694,8] := 2.0;
   DATA[694,9] := 2.0;
   DATA[694,10] := 2.0;
   DATA[694,11] := 19.72277;
   DATA[694,12] := 2.210678;
   DATA[694,13] := 989.3698;
   DATA[694,14] := 1.0;
   DATA[694,15] := 2.0;
   DATA[694,16] := 1.0;
   DATA[694,17] := 1.0;
   DATA[694,18] := 1.0;
   DATA[694,19] := 2.0;
   DATA[694,20] := 148.808;
   DATA[694,21] := 155.5499;
   DATA[694,22] := 1.719284;
   DATA[694,23] := 998.7054;
   DATA[694,24] := 2.0;
   DATA[694,25] := 2.0;
   DATA[694,26] := 7.878942;
   DATA[694,27] := 144.7578;
   DATA[694,28] := 263.1377;
   DATA[694,29] := 12.11228;
   DATA[694,30] := 1.729172;
   DATA[694,31] := 1.281542;
   DATA[694,32] := 0.7352687;
   DATA[694,33] := 0.3064407;
   DATA[694,34] := 2.0;
   DATA[694,35] := 251.0734;
   DATA[694,36] := 1.69801;
   DATA[694,37] := 189.8872;
   DATA[694,38] := 0.000128152;
   DATA[694,39] := 1.0;
   DATA[695,0] := 2.573744;
   DATA[695,1] := 538.0375;
   DATA[695,2] := 2.0;
   DATA[695,3] := 2.0;
   DATA[695,4] := 262.1764;
   DATA[695,5] := 8.395475;
   DATA[695,6] := 327.7108;
   DATA[695,7] := 2.439881;
   DATA[695,8] := 2.0;
   DATA[695,9] := 2.0;
   DATA[695,10] := 2.0;
   DATA[695,11] := 19.63954;
   DATA[695,12] := 2.210166;
   DATA[695,13] := 989.0493;
   DATA[695,14] := 1.0;
   DATA[695,15] := 2.0;
   DATA[695,16] := 1.0;
   DATA[695,17] := 1.0;
   DATA[695,18] := 1.0;
   DATA[695,19] := 2.0;
   DATA[695,20] := 148.808;
   DATA[695,21] := 155.6524;
   DATA[695,22] := 1.719284;
   DATA[695,23] := 998.8208;
   DATA[695,24] := 2.0;
   DATA[695,25] := 2.0;
   DATA[695,26] := 7.878942;
   DATA[695,27] := 144.8347;
   DATA[695,28] := 263.2658;
   DATA[695,29] := 12.11228;
   DATA[695,30] := 1.728019;
   DATA[695,31] := 1.281542;
   DATA[695,32] := 0.7352687;
   DATA[695,33] := 0.3064407;
   DATA[695,34] := 2.0;
   DATA[695,35] := 251.0734;
   DATA[695,36] := 1.730048;
   DATA[695,37] := 189.727;
   DATA[695,38] := 0.000128152;
   DATA[695,39] := 1.0;
   DATA[696,0] := 2.551324;
   DATA[696,1] := 537.8021;
   DATA[696,2] := 2.0;
   DATA[696,3] := 2.0;
   DATA[696,4] := 262.1764;
   DATA[696,5] := 8.395475;
   DATA[696,6] := 327.7108;
   DATA[696,7] := 2.439881;
   DATA[696,8] := 2.0;
   DATA[696,9] := 2.0;
   DATA[696,10] := 2.0;
   DATA[696,11] := 19.63954;
   DATA[696,12] := 2.210166;
   DATA[696,13] := 988.8891;
   DATA[696,14] := 1.0;
   DATA[696,15] := 2.0;
   DATA[696,16] := 1.0;
   DATA[696,17] := 1.0;
   DATA[696,18] := 1.0;
   DATA[696,19] := 2.0;
   DATA[696,20] := 148.808;
   DATA[696,21] := 155.6524;
   DATA[696,22] := 1.718515;
   DATA[696,23] := 998.5516;
   DATA[696,24] := 2.0;
   DATA[696,25] := 2.0;
   DATA[696,26] := 7.878942;
   DATA[696,27] := 144.8347;
   DATA[696,28] := 263.362;
   DATA[696,29] := 12.11228;
   DATA[696,30] := 1.728019;
   DATA[696,31] := 1.281542;
   DATA[696,32] := 0.7352687;
   DATA[696,33] := 0.3064407;
   DATA[696,34] := 2.0;
   DATA[696,35] := 251.0734;
   DATA[696,36] := 1.730048;
   DATA[696,37] := 189.727;
   DATA[696,38] := 0.000128152;
   DATA[696,39] := 1.0;
   DATA[697,0] := 2.539154;
   DATA[697,1] := 537.8413;
   DATA[697,2] := 2.0;
   DATA[697,3] := 2.0;
   DATA[697,4] := 262.1764;
   DATA[697,5] := 8.395475;
   DATA[697,6] := 327.7108;
   DATA[697,7] := 2.441803;
   DATA[697,8] := 2.0;
   DATA[697,9] := 2.0;
   DATA[697,10] := 2.0;
   DATA[697,11] := 19.63954;
   DATA[697,12] := 2.210166;
   DATA[697,13] := 988.8491;
   DATA[697,14] := 1.0;
   DATA[697,15] := 2.0;
   DATA[697,16] := 1.0;
   DATA[697,17] := 1.0;
   DATA[697,18] := 1.0;
   DATA[697,19] := 2.0;
   DATA[697,20] := 148.808;
   DATA[697,21] := 155.7037;
   DATA[697,22] := 1.718515;
   DATA[697,23] := 998.8208;
   DATA[697,24] := 2.0;
   DATA[697,25] := 2.0;
   DATA[697,26] := 7.878942;
   DATA[697,27] := 144.8347;
   DATA[697,28] := 263.362;
   DATA[697,29] := 12.11228;
   DATA[697,30] := 1.728019;
   DATA[697,31] := 1.281542;
   DATA[697,32] := 0.7352687;
   DATA[697,33] := 0.3064407;
   DATA[697,34] := 2.0;
   DATA[697,35] := 251.0734;
   DATA[697,36] := 1.730048;
   DATA[697,37] := 189.727;
   DATA[697,38] := 0.000128152;
   DATA[697,39] := 1.0;
   DATA[698,0] := 2.518656;
   DATA[698,1] := 538.1553;
   DATA[698,2] := 2.0;
   DATA[698,3] := 2.0;
   DATA[698,4] := 262.1764;
   DATA[698,5] := 8.395475;
   DATA[698,6] := 327.7108;
   DATA[698,7] := 2.442444;
   DATA[698,8] := 2.0;
   DATA[698,9] := 2.0;
   DATA[698,10] := 2.0;
   DATA[698,11] := 19.60433;
   DATA[698,12] := 2.210166;
   DATA[698,13] := 988.9692;
   DATA[698,14] := 1.0;
   DATA[698,15] := 2.0;
   DATA[698,16] := 1.0;
   DATA[698,17] := 1.0;
   DATA[698,18] := 1.0;
   DATA[698,19] := 2.0;
   DATA[698,20] := 148.808;
   DATA[698,21] := 155.7037;
   DATA[698,22] := 1.718515;
   DATA[698,23] := 998.7439;
   DATA[698,24] := 2.0;
   DATA[698,25] := 2.0;
   DATA[698,26] := 7.878942;
   DATA[698,27] := 144.8347;
   DATA[698,28] := 263.362;
   DATA[698,29] := 12.11228;
   DATA[698,30] := 1.728019;
   DATA[698,31] := 1.275266;
   DATA[698,32] := 0.7352687;
   DATA[698,33] := 0.3064407;
   DATA[698,34] := 2.0;
   DATA[698,35] := 250.9453;
   DATA[698,36] := 1.730048;
   DATA[698,37] := 189.727;
   DATA[698,38] := 0.000128152;
   DATA[698,39] := 1.0;
   DATA[699,0] := 2.497198;
   DATA[699,1] := 538.3908;
   DATA[699,2] := 2.0;
   DATA[699,3] := 2.0;
   DATA[699,4] := 262.1764;
   DATA[699,5] := 8.395475;
   DATA[699,6] := 327.7108;
   DATA[699,7] := 2.442444;
   DATA[699,8] := 2.0;
   DATA[699,9] := 2.0;
   DATA[699,10] := 2.0;
   DATA[699,11] := 19.57552;
   DATA[699,12] := 2.210166;
   DATA[699,13] := 988.6888;
   DATA[699,14] := 1.0;
   DATA[699,15] := 2.0;
   DATA[699,16] := 1.0;
   DATA[699,17] := 1.0;
   DATA[699,18] := 1.0;
   DATA[699,19] := 2.0;
   DATA[699,20] := 148.808;
   DATA[699,21] := 155.7037;
   DATA[699,22] := 1.717489;
   DATA[699,23] := 999.0515;
   DATA[699,24] := 2.0;
   DATA[699,25] := 2.0;
   DATA[699,26] := 7.878942;
   DATA[699,27] := 144.8347;
   DATA[699,28] := 263.362;
   DATA[699,29] := 12.11228;
   DATA[699,30] := 1.728019;
   DATA[699,31] := 1.277187;
   DATA[699,32] := 0.7352687;
   DATA[699,33] := 0.3064407;
   DATA[699,34] := 2.0;
   DATA[699,35] := 250.9453;
   DATA[699,36] := 1.730048;
   DATA[699,37] := 189.727;
   DATA[699,38] := 0.000128152;
   DATA[699,39] := 1.0;
   DATA[700,0] := 2.485988;
   DATA[700,1] := 538.2731;
   DATA[700,2] := 2.0;
   DATA[700,3] := 2.0;
   DATA[700,4] := 262.1764;
   DATA[700,5] := 8.395475;
   DATA[700,6] := 327.7108;
   DATA[700,7] := 2.442444;
   DATA[700,8] := 2.0;
   DATA[700,9] := 2.0;
   DATA[700,10] := 2.0;
   DATA[700,11] := 19.57552;
   DATA[700,12] := 2.210166;
   DATA[700,13] := 988.5687;
   DATA[700,14] := 1.0;
   DATA[700,15] := 2.0;
   DATA[700,16] := 1.0;
   DATA[700,17] := 1.0;
   DATA[700,18] := 1.0;
   DATA[700,19] := 2.0;
   DATA[700,20] := 148.808;
   DATA[700,21] := 155.7037;
   DATA[700,22] := 1.717489;
   DATA[700,23] := 999.0131;
   DATA[700,24] := 2.0;
   DATA[700,25] := 2.0;
   DATA[700,26] := 7.878942;
   DATA[700,27] := 144.8347;
   DATA[700,28] := 263.362;
   DATA[700,29] := 12.11228;
   DATA[700,30] := 1.728019;
   DATA[700,31] := 1.271679;
   DATA[700,32] := 0.7352687;
   DATA[700,33] := 0.3064407;
   DATA[700,34] := 2.0;
   DATA[700,35] := 250.9453;
   DATA[700,36] := 1.730048;
   DATA[700,37] := 189.727;
   DATA[700,38] := 0.000128152;
   DATA[700,39] := 1.0;
   DATA[701,0] := 2.471896;
   DATA[701,1] := 537.9983;
   DATA[701,2] := 2.0;
   DATA[701,3] := 2.0;
   DATA[701,4] := 262.1764;
   DATA[701,5] := 8.395475;
   DATA[701,6] := 327.7108;
   DATA[701,7] := 2.442444;
   DATA[701,8] := 2.0;
   DATA[701,9] := 2.0;
   DATA[701,10] := 2.0;
   DATA[701,11] := 19.57552;
   DATA[701,12] := 2.211447;
   DATA[701,13] := 988.088;
   DATA[701,14] := 1.0;
   DATA[701,15] := 2.0;
   DATA[701,16] := 1.0;
   DATA[701,17] := 1.0;
   DATA[701,18] := 1.0;
   DATA[701,19] := 2.0;
   DATA[701,20] := 148.808;
   DATA[701,21] := 155.7037;
   DATA[701,22] := 1.717489;
   DATA[701,23] := 999.2053;
   DATA[701,24] := 2.0;
   DATA[701,25] := 2.0;
   DATA[701,26] := 7.878942;
   DATA[701,27] := 144.8347;
   DATA[701,28] := 263.362;
   DATA[701,29] := 12.11228;
   DATA[701,30] := 1.728019;
   DATA[701,31] := 1.271551;
   DATA[701,32] := 0.7352687;
   DATA[701,33] := 0.3069532;
   DATA[701,34] := 2.0;
   DATA[701,35] := 250.9453;
   DATA[701,36] := 1.730048;
   DATA[701,37] := 189.727;
   DATA[701,38] := 0.000128152;
   DATA[701,39] := 1.0;
   DATA[702,0] := 2.45428;
   DATA[702,1] := 537.959;
   DATA[702,2] := 2.0;
   DATA[702,3] := 2.0;
   DATA[702,4] := 262.1764;
   DATA[702,5] := 8.395475;
   DATA[702,6] := 327.7108;
   DATA[702,7] := 2.442444;
   DATA[702,8] := 2.0;
   DATA[702,9] := 2.0;
   DATA[702,10] := 2.0;
   DATA[702,11] := 19.5371;
   DATA[702,12] := 2.212215;
   DATA[702,13] := 987.6474;
   DATA[702,14] := 1.0;
   DATA[702,15] := 2.0;
   DATA[702,16] := 1.0;
   DATA[702,17] := 1.0;
   DATA[702,18] := 1.0;
   DATA[702,19] := 2.0;
   DATA[702,20] := 148.808;
   DATA[702,21] := 155.7037;
   DATA[702,22] := 1.717489;
   DATA[702,23] := 998.8977;
   DATA[702,24] := 2.0;
   DATA[702,25] := 2.0;
   DATA[702,26] := 7.878942;
   DATA[702,27] := 144.8347;
   DATA[702,28] := 263.2979;
   DATA[702,29] := 12.11228;
   DATA[702,30] := 1.728019;
   DATA[702,31] := 1.287947;
   DATA[702,32] := 0.7352687;
   DATA[702,33] := 0.3069532;
   DATA[702,34] := 2.0;
   DATA[702,35] := 250.9453;
   DATA[702,36] := 1.730048;
   DATA[702,37] := 189.727;
   DATA[702,38] := 0.000128152;
   DATA[702,39] := 1.0;
   DATA[703,0] := 2.443071;
   DATA[703,1] := 538.0375;
   DATA[703,2] := 2.0;
   DATA[703,3] := 2.0;
   DATA[703,4] := 262.1764;
   DATA[703,5] := 8.395475;
   DATA[703,6] := 327.7108;
   DATA[703,7] := 2.442444;
   DATA[703,8] := 2.0;
   DATA[703,9] := 2.0;
   DATA[703,10] := 2.0;
   DATA[703,11] := 19.5243;
   DATA[703,12] := 2.212215;
   DATA[703,13] := 987.5673;
   DATA[703,14] := 1.0;
   DATA[703,15] := 2.0;
   DATA[703,16] := 1.0;
   DATA[703,17] := 1.0;
   DATA[703,18] := 1.0;
   DATA[703,19] := 2.0;
   DATA[703,20] := 148.808;
   DATA[703,21] := 155.7037;
   DATA[703,22] := 1.717489;
   DATA[703,23] := 999.3976;
   DATA[703,24] := 2.0;
   DATA[703,25] := 2.0;
   DATA[703,26] := 7.878942;
   DATA[703,27] := 144.8347;
   DATA[703,28] := 263.1056;
   DATA[703,29] := 12.11228;
   DATA[703,30] := 1.729428;
   DATA[703,31] := 1.299219;
   DATA[703,32] := 0.7352687;
   DATA[703,33] := 0.3069532;
   DATA[703,34] := 2.0;
   DATA[703,35] := 250.9453;
   DATA[703,36] := 1.730048;
   DATA[703,37] := 189.727;
   DATA[703,38] := 0.000128152;
   DATA[703,39] := 1.0;
   DATA[704,0] := 2.431221;
   DATA[704,1] := 537.9983;
   DATA[704,2] := 2.0;
   DATA[704,3] := 2.0;
   DATA[704,4] := 262.1764;
   DATA[704,5] := 8.395475;
   DATA[704,6] := 327.7108;
   DATA[704,7] := 2.441034;
   DATA[704,8] := 2.0;
   DATA[704,9] := 2.0;
   DATA[704,10] := 2.0;
   DATA[704,11] := 19.55951;
   DATA[704,12] := 2.210294;
   DATA[704,13] := 987.8477;
   DATA[704,14] := 1.0;
   DATA[704,15] := 2.0;
   DATA[704,16] := 1.0;
   DATA[704,17] := 1.0;
   DATA[704,18] := 1.0;
   DATA[704,19] := 2.0;
   DATA[704,20] := 148.808;
   DATA[704,21] := 155.7037;
   DATA[704,22] := 1.720309;
   DATA[704,23] := 999.4745;
   DATA[704,24] := 2.0;
   DATA[704,25] := 2.0;
   DATA[704,26] := 7.878942;
   DATA[704,27] := 144.8347;
   DATA[704,28] := 263.1056;
   DATA[704,29] := 12.11228;
   DATA[704,30] := 1.731095;
   DATA[704,31] := 1.30178;
   DATA[704,32] := 0.7352687;
   DATA[704,33] := 0.3069532;
   DATA[704,34] := 2.0;
   DATA[704,35] := 250.9453;
   DATA[704,36] := 1.730048;
   DATA[704,37] := 189.727;
   DATA[704,38] := 0.000128152;
   DATA[704,39] := 1.0;
   DATA[705,0] := 2.429619;
   DATA[705,1] := 537.3702;
   DATA[705,2] := 2.0;
   DATA[705,3] := 2.0;
   DATA[705,4] := 262.1764;
   DATA[705,5] := 8.395475;
   DATA[705,6] := 327.7108;
   DATA[705,7] := 2.439753;
   DATA[705,8] := 2.0;
   DATA[705,9] := 2.0;
   DATA[705,10] := 2.0;
   DATA[705,11] := 19.59793;
   DATA[705,12] := 2.210294;
   DATA[705,13] := 987.9678;
   DATA[705,14] := 1.0;
   DATA[705,15] := 2.0;
   DATA[705,16] := 1.0;
   DATA[705,17] := 1.0;
   DATA[705,18] := 1.0;
   DATA[705,19] := 2.0;
   DATA[705,20] := 148.808;
   DATA[705,21] := 155.7037;
   DATA[705,22] := 1.720309;
   DATA[705,23] := 999.7821;
   DATA[705,24] := 2.0;
   DATA[705,25] := 2.0;
   DATA[705,26] := 7.878942;
   DATA[705,27] := 144.8347;
   DATA[705,28] := 263.1056;
   DATA[705,29] := 12.11228;
   DATA[705,30] := 1.731095;
   DATA[705,31] := 1.30178;
   DATA[705,32] := 0.7352687;
   DATA[705,33] := 0.3068891;
   DATA[705,34] := 2.0;
   DATA[705,35] := 250.9453;
   DATA[705,36] := 1.730048;
   DATA[705,37] := 189.727;
   DATA[705,38] := 0.000128152;
   DATA[705,39] := 1.0;
   DATA[706,0] := 2.436345;
   DATA[706,1] := 537.4488;
   DATA[706,2] := 2.0;
   DATA[706,3] := 2.0;
   DATA[706,4] := 262.1764;
   DATA[706,5] := 8.395475;
   DATA[706,6] := 327.7108;
   DATA[706,7] := 2.439753;
   DATA[706,8] := 2.0;
   DATA[706,9] := 2.0;
   DATA[706,10] := 2.0;
   DATA[706,11] := 19.65235;
   DATA[706,12] := 2.210294;
   DATA[706,13] := 987.6875;
   DATA[706,14] := 1.0;
   DATA[706,15] := 2.0;
   DATA[706,16] := 1.0;
   DATA[706,17] := 1.0;
   DATA[706,18] := 1.0;
   DATA[706,19] := 2.0;
   DATA[706,20] := 148.808;
   DATA[706,21] := 155.7037;
   DATA[706,22] := 1.718515;
   DATA[706,23] := 999.3976;
   DATA[706,24] := 2.0;
   DATA[706,25] := 2.0;
   DATA[706,26] := 7.878942;
   DATA[706,27] := 144.7065;
   DATA[706,28] := 263.1056;
   DATA[706,29] := 12.11228;
   DATA[706,30] := 1.731095;
   DATA[706,31] := 1.292174;
   DATA[706,32] := 0.7352687;
   DATA[706,33] := 0.3063127;
   DATA[706,34] := 2.0;
   DATA[706,35] := 250.9453;
   DATA[706,36] := 1.730048;
   DATA[706,37] := 189.727;
   DATA[706,38] := 0.000128152;
   DATA[706,39] := 1.0;
   DATA[707,0] := 2.479903;
   DATA[707,1] := 537.2133;
   DATA[707,2] := 2.0;
   DATA[707,3] := 2.0;
   DATA[707,4] := 262.1764;
   DATA[707,5] := 8.395475;
   DATA[707,6] := 327.7108;
   DATA[707,7] := 2.438471;
   DATA[707,8] := 2.0;
   DATA[707,9] := 2.0;
   DATA[707,10] := 2.0;
   DATA[707,11] := 19.65235;
   DATA[707,12] := 2.210294;
   DATA[707,13] := 987.8477;
   DATA[707,14] := 1.0;
   DATA[707,15] := 2.0;
   DATA[707,16] := 1.0;
   DATA[707,17] := 1.0;
   DATA[707,18] := 1.0;
   DATA[707,19] := 2.0;
   DATA[707,20] := 148.808;
   DATA[707,21] := 155.7037;
   DATA[707,22] := 1.71813;
   DATA[707,23] := 999.8206;
   DATA[707,24] := 2.0;
   DATA[707,25] := 2.0;
   DATA[707,26] := 7.878942;
   DATA[707,27] := 144.7065;
   DATA[707,28] := 263.1056;
   DATA[707,29] := 12.11228;
   DATA[707,30] := 1.731095;
   DATA[707,31] := 1.283848;
   DATA[707,32] := 0.7352687;
   DATA[707,33] := 0.3063127;
   DATA[707,34] := 2.0;
   DATA[707,35] := 250.9453;
   DATA[707,36] := 1.730048;
   DATA[707,37] := 189.727;
   DATA[707,38] := 0.000128152;
   DATA[707,39] := 1.0;
   DATA[708,0] := 2.528905;
   DATA[708,1] := 537.4488;
   DATA[708,2] := 2.0;
   DATA[708,3] := 2.0;
   DATA[708,4] := 262.1764;
   DATA[708,5] := 8.395475;
   DATA[708,6] := 327.7108;
   DATA[708,7] := 2.437318;
   DATA[708,8] := 2.0;
   DATA[708,9] := 2.0;
   DATA[708,10] := 2.0;
   DATA[708,11] := 19.65235;
   DATA[708,12] := 2.210294;
   DATA[708,13] := 987.8878;
   DATA[708,14] := 1.0;
   DATA[708,15] := 2.0;
   DATA[708,16] := 1.0;
   DATA[708,17] := 1.0;
   DATA[708,18] := 1.0;
   DATA[708,19] := 1.0;
   DATA[708,20] := 148.808;
   DATA[708,21] := 155.7037;
   DATA[708,22] := 1.718002;
   DATA[708,23] := 999.8975;
   DATA[708,24] := 2.0;
   DATA[708,25] := 2.0;
   DATA[708,26] := 7.878942;
   DATA[708,27] := 144.7065;
   DATA[708,28] := 263.1056;
   DATA[708,29] := 12.11228;
   DATA[708,30] := 1.731095;
   DATA[708,31] := 1.282183;
   DATA[708,32] := 0.7352687;
   DATA[708,33] := 0.3063127;
   DATA[708,34] := 2.0;
   DATA[708,35] := 250.9453;
   DATA[708,36] := 1.730048;
   DATA[708,37] := 189.727;
   DATA[708,38] := 0.000128152;
   DATA[708,39] := 1.0;
   DATA[709,0] := 2.571182;
   DATA[709,1] := 537.0955;
   DATA[709,2] := 2.0;
   DATA[709,3] := 2.0;
   DATA[709,4] := 262.1764;
   DATA[709,5] := 8.395475;
   DATA[709,6] := 327.7108;
   DATA[709,7] := 2.437318;
   DATA[709,8] := 2.0;
   DATA[709,9] := 2.0;
   DATA[709,10] := 2.0;
   DATA[709,11] := 19.37064;
   DATA[709,12] := 2.210294;
   DATA[709,13] := 988.088;
   DATA[709,14] := 1.0;
   DATA[709,15] := 2.0;
   DATA[709,16] := 1.0;
   DATA[709,17] := 1.0;
   DATA[709,18] := 1.0;
   DATA[709,19] := 1.0;
   DATA[709,20] := 148.808;
   DATA[709,21] := 155.7037;
   DATA[709,22] := 1.718002;
   DATA[709,23] := 1000.205;
   DATA[709,24] := 2.0;
   DATA[709,25] := 2.0;
   DATA[709,26] := 7.878942;
   DATA[709,27] := 144.7065;
   DATA[709,28] := 263.1056;
   DATA[709,29] := 12.11228;
   DATA[709,30] := 1.731095;
   DATA[709,31] := 1.299603;
   DATA[709,32] := 0.7352687;
   DATA[709,33] := 0.3063127;
   DATA[709,34] := 2.0;
   DATA[709,35] := 250.9453;
   DATA[709,36] := 1.730048;
   DATA[709,37] := 189.727;
   DATA[709,38] := 0.000128152;
   DATA[709,39] := 1.0;
   DATA[710,0] := 2.601608;
   DATA[710,1] := 536.5067;
   DATA[710,2] := 2.0;
   DATA[710,3] := 2.0;
   DATA[710,4] := 262.1764;
   DATA[710,5] := 8.395475;
   DATA[710,6] := 327.7108;
   DATA[710,7] := 2.437318;
   DATA[710,8] := 2.0;
   DATA[710,9] := 2.0;
   DATA[710,10] := 2.0;
   DATA[710,11] := 18.27582;
   DATA[710,12] := 2.20171;
   DATA[710,13] := 987.8878;
   DATA[710,14] := 1.0;
   DATA[710,16] := 1.0;
   DATA[710,17] := 1.0;
   DATA[710,18] := 1.0;
   DATA[710,19] := 1.0;
   DATA[710,20] := 148.808;
   DATA[710,21] := 155.7037;
   DATA[710,22] := 1.718002;
   DATA[710,23] := 1000.051;
   DATA[710,24] := 2.0;
   DATA[710,25] := 2.0;
   DATA[710,26] := 7.878942;
   DATA[710,27] := 144.7065;
   DATA[710,28] := 263.1056;
   DATA[710,29] := 12.11228;
   DATA[710,30] := 1.731095;
   DATA[710,31] := 1.301012;
   DATA[710,32] := 0.7352687;
   DATA[710,33] := 0.3066329;
   DATA[710,34] := 2.0;
   DATA[710,35] := 251.1215;
   DATA[710,36] := 1.730048;
   DATA[710,37] := 189.7751;
   DATA[710,38] := 0.000128152;
   DATA[710,39] := 1.0;
   DATA[711,0] := 2.637799;
   DATA[711,1] := 536.2319;
   DATA[711,2] := 2.0;
   DATA[711,3] := 2.0;
   DATA[711,4] := 262.1764;
   DATA[711,5] := 8.395475;
   DATA[711,6] := 327.7108;
   DATA[711,7] := 2.43924;
   DATA[711,8] := 2.0;
   DATA[711,9] := 2.0;
   DATA[711,10] := 2.0;
   DATA[711,11] := 16.38389;
   DATA[711,12] := 2.124075;
   DATA[711,13] := 988.4084;
   DATA[711,14] := 1.0;
   DATA[711,16] := 1.0;
   DATA[711,17] := 1.0;
   DATA[711,18] := 1.0;
   DATA[711,19] := 1.0;
   DATA[711,20] := 148.808;
   DATA[711,21] := 155.7037;
   DATA[711,22] := 1.718002;
   DATA[711,23] := 1000.205;
   DATA[711,24] := 2.0;
   DATA[711,25] := 2.0;
   DATA[711,26] := 7.878942;
   DATA[711,27] := 144.7065;
   DATA[711,28] := 263.1056;
   DATA[711,29] := 12.11228;
   DATA[711,30] := 1.731095;
   DATA[711,31] := 1.297041;
   DATA[711,32] := 0.7352687;
   DATA[711,33] := 0.3066329;
   DATA[711,34] := 2.0;
   DATA[711,35] := 251.2657;
   DATA[711,36] := 1.730048;
   DATA[711,37] := 189.9673;
   DATA[711,38] := 0.000128152;
   DATA[711,39] := 1.0;
   DATA[712,0] := 2.66214;
   DATA[712,1] := 536.7029;
   DATA[712,2] := 2.0;
   DATA[712,3] := 2.0;
   DATA[712,4] := 262.1764;
   DATA[712,5] := 8.395475;
   DATA[712,6] := 327.7108;
   DATA[712,7] := 2.440265;
   DATA[712,8] := 2.0;
   DATA[712,9] := 2.0;
   DATA[712,10] := 2.0;
   DATA[712,11] := 13.86773;
   DATA[712,12] := 1.967524;
   DATA[712,13] := 988.6087;
   DATA[712,14] := 1.0;
   DATA[712,16] := 1.0;
   DATA[712,17] := 1.0;
   DATA[712,18] := 1.0;
   DATA[712,19] := 1.0;
   DATA[712,20] := 148.808;
   DATA[712,21] := 155.7037;
   DATA[712,22] := 1.718002;
   DATA[712,23] := 1000.282;
   DATA[712,24] := 2.0;
   DATA[712,25] := 2.0;
   DATA[712,26] := 7.878942;
   DATA[712,27] := 144.7065;
   DATA[712,28] := 263.1056;
   DATA[712,29] := 12.11228;
   DATA[712,30] := 1.731095;
   DATA[712,31] := 1.297682;
   DATA[712,32] := 0.7352687;
   DATA[712,33] := 0.3066329;
   DATA[712,34] := 2.0;
   DATA[712,35] := 251.2657;
   DATA[712,36] := 1.730048;
   DATA[712,37] := 189.9833;
   DATA[712,38] := 0.000128152;
   DATA[712,39] := 1.0;
   DATA[713,0] := 2.662781;
   DATA[713,1] := 536.8207;
   DATA[713,2] := 2.0;
   DATA[713,3] := 2.0;
   DATA[713,4] := 262.1764;
   DATA[713,5] := 8.395475;
   DATA[713,6] := 327.7108;
   DATA[713,7] := 2.440265;
   DATA[713,8] := 2.0;
   DATA[713,9] := 2.0;
   DATA[713,10] := 2.0;
   DATA[713,11] := 11.11787;
   DATA[713,12] := 1.669026;
   DATA[713,13] := 988.8491;
   DATA[713,14] := 1.0;
   DATA[713,16] := 1.0;
   DATA[713,17] := 1.0;
   DATA[713,18] := 1.0;
   DATA[713,19] := 1.0;
   DATA[713,20] := 148.808;
   DATA[713,21] := 155.7037;
   DATA[713,22] := 1.719668;
   DATA[713,23] := 1000.09;
   DATA[713,24] := 2.0;
   DATA[713,25] := 2.0;
   DATA[713,26] := 7.878942;
   DATA[713,27] := 144.7065;
   DATA[713,28] := 263.1056;
   DATA[713,29] := 12.11228;
   DATA[713,30] := 1.731095;
   DATA[713,31] := 1.282183;
   DATA[713,32] := 0.7352687;
   DATA[713,33] := 0.3066329;
   DATA[713,34] := 2.0;
   DATA[713,35] := 251.2657;
   DATA[713,36] := 1.730048;
   DATA[713,37] := 189.9833;
   DATA[713,38] := 0.000128152;
   DATA[713,39] := 1.0;
   DATA[714,0] := 2.649009;
   DATA[714,1] := 536.8207;
   DATA[714,2] := 2.0;
   DATA[714,3] := 2.0;
   DATA[714,4] := 262.1764;
   DATA[714,5] := 8.395475;
   DATA[714,6] := 327.7108;
   DATA[714,7] := 2.440265;
   DATA[714,8] := 2.0;
   DATA[714,9] := 2.0;
   DATA[714,10] := 2.0;
   DATA[714,11] := 9.027467;
   DATA[714,12] := 1.351568;
   DATA[714,13] := 988.8491;
   DATA[714,14] := 1.0;
   DATA[714,16] := 1.0;
   DATA[714,17] := 1.0;
   DATA[714,18] := 1.0;
   DATA[714,19] := 1.0;
   DATA[714,20] := 148.808;
   DATA[714,21] := 155.7037;
   DATA[714,22] := 1.721975;
   DATA[714,23] := 1000.013;
   DATA[714,24] := 2.0;
   DATA[714,25] := 2.0;
   DATA[714,26] := 7.878942;
   DATA[714,27] := 144.7065;
   DATA[714,28] := 263.1056;
   DATA[714,29] := 12.11228;
   DATA[714,30] := 1.731095;
   DATA[714,31] := 1.281798;
   DATA[714,32] := 0.7352687;
   DATA[714,33] := 0.3066329;
   DATA[714,34] := 2.0;
   DATA[714,35] := 251.2657;
   DATA[714,36] := 1.730048;
   DATA[714,37] := 189.9833;
   DATA[714,38] := 0.000128152;
   DATA[714,39] := 1.0;
   DATA[715,0] := 2.649009;
   DATA[715,1] := 536.8207;
   DATA[715,2] := 2.0;
   DATA[715,3] := 2.0;
   DATA[715,4] := 262.1764;
   DATA[715,5] := 8.395475;
   DATA[715,6] := 327.7108;
   DATA[715,7] := 2.440265;
   DATA[715,8] := 2.0;
   DATA[715,9] := 2.0;
   DATA[715,10] := 2.0;
   DATA[715,11] := 9.027467;
   DATA[715,12] := 1.351568;
   DATA[715,13] := 988.8491;
   DATA[715,14] := 1.0;
   DATA[715,16] := 1.0;
   DATA[715,17] := 1.0;
   DATA[715,18] := 1.0;
   DATA[715,19] := 1.0;
   DATA[715,20] := 148.808;
   DATA[715,21] := 155.7037;
   DATA[715,22] := 1.721975;
   DATA[715,23] := 1000.013;
   DATA[715,24] := 2.0;
   DATA[715,25] := 2.0;
   DATA[715,26] := 7.878942;
   DATA[715,27] := 144.7065;
   DATA[715,28] := 263.1056;
   DATA[715,29] := 12.11228;
   DATA[715,30] := 1.731095;
   DATA[715,31] := 1.281798;
   DATA[715,32] := 0.7352687;
   DATA[715,33] := 0.3066329;
   DATA[715,34] := 2.0;
   DATA[715,35] := 251.2657;
   DATA[715,36] := 1.730048;
   DATA[715,37] := 189.9833;
   DATA[715,38] := 0.000128152;
   DATA[715,39] := 1.0;
   DATA[716,0] := 2.620184;
   DATA[716,1] := 536.2712;
   DATA[716,2] := 2.0;
   DATA[716,3] := 2.0;
   DATA[716,4] := 262.1764;
   DATA[716,5] := 8.395475;
   DATA[716,6] := 327.7108;
   DATA[716,7] := 2.441419;
   DATA[716,8] := 2.0;
   DATA[716,9] := 2.0;
   DATA[716,10] := 2.0;
   DATA[716,11] := 7.122735;
   DATA[716,12] := 0.974538;
   DATA[716,13] := 988.809;
   DATA[716,14] := 1.0;
   DATA[716,16] := 1.0;
   DATA[716,17] := 1.0;
   DATA[716,18] := 1.0;
   DATA[716,19] := 1.0;
   DATA[716,20] := 148.808;
   DATA[716,21] := 155.7037;
   DATA[716,22] := 1.724153;
   DATA[716,23] := 1000.244;
   DATA[716,24] := 2.0;
   DATA[716,25] := 2.0;
   DATA[716,26] := 7.878942;
   DATA[716,27] := 144.7065;
   DATA[716,28] := 263.1056;
   DATA[716,29] := 12.11228;
   DATA[716,30] := 1.731095;
   DATA[716,31] := 1.281798;
   DATA[716,32] := 0.7352687;
   DATA[716,33] := 0.3066329;
   DATA[716,34] := 2.0;
   DATA[716,35] := 251.3458;
   DATA[716,36] := 1.730048;
   DATA[716,37] := 189.9833;
   DATA[716,38] := 0.000128152;
   DATA[716,39] := 1.0;
   DATA[717,0] := 2.612497;
   DATA[717,1] := 535.8002;
   DATA[717,2] := 2.0;
   DATA[717,3] := 2.0;
   DATA[717,4] := 262.1764;
   DATA[717,5] := 8.395475;
   DATA[717,6] := 327.7108;
   DATA[717,7] := 2.44206;
   DATA[717,8] := 2.0;
   DATA[717,9] := 2.0;
   DATA[717,10] := 2.0;
   DATA[717,11] := 5.045137;
   DATA[717,12] := 0.5084713;
   DATA[717,13] := 988.809;
   DATA[717,14] := 1.0;
   DATA[717,16] := 1.0;
   DATA[717,17] := 1.0;
   DATA[717,18] := 1.0;
   DATA[717,19] := 1.0;
   DATA[717,20] := 148.808;
   DATA[717,21] := 155.7037;
   DATA[717,22] := 1.724153;
   DATA[717,23] := 1000.244;
   DATA[717,24] := 2.0;
   DATA[717,25] := 2.0;
   DATA[717,26] := 7.878942;
   DATA[717,27] := 144.7065;
   DATA[717,28] := 263.1056;
   DATA[717,29] := 12.11228;
   DATA[717,30] := 1.731095;
   DATA[717,31] := 1.271935;
   DATA[717,32] := 0.7352687;
   DATA[717,33] := 0.3066329;
   DATA[717,34] := 2.0;
   DATA[717,35] := 251.3618;
   DATA[717,36] := 1.730048;
   DATA[717,37] := 190.1275;
   DATA[717,38] := 0.000128152;
   DATA[717,39] := 1.0;
   DATA[718,0] := 2.612497;
   DATA[718,1] := 535.8787;
   DATA[718,2] := 2.0;
   DATA[718,3] := 2.0;
   DATA[718,4] := 262.1764;
   DATA[718,5] := 8.395475;
   DATA[718,6] := 327.7108;
   DATA[718,7] := 2.44206;
   DATA[718,8] := 2.0;
   DATA[718,9] := 2.0;
   DATA[718,10] := 2.0;
   DATA[718,11] := 4.324861;
   DATA[718,12] := 0.356532;
   DATA[718,13] := 989.0493;
   DATA[718,14] := 1.0;
   DATA[718,15] := 1.0;
   DATA[718,16] := 1.0;
   DATA[718,17] := 1.0;
   DATA[718,18] := 1.0;
   DATA[718,19] := 1.0;
   DATA[718,20] := 148.808;
   DATA[718,21] := 155.7037;
   DATA[718,22] := 1.724153;
   DATA[718,23] := 1000.282;
   DATA[718,24] := 2.0;
   DATA[718,25] := 2.0;
   DATA[718,26] := 7.878942;
   DATA[718,27] := 144.7065;
   DATA[718,28] := 263.1056;
   DATA[718,29] := 12.11228;
   DATA[718,30] := 1.731095;
   DATA[718,31] := 1.280005;
   DATA[718,32] := 0.7352687;
   DATA[718,33] := 0.3066329;
   DATA[718,34] := 2.0;
   DATA[718,35] := 251.3618;
   DATA[718,36] := 1.730048;
   DATA[718,37] := 190.1275;
   DATA[718,38] := 0.000128152;
   DATA[718,39] := 1.0;
   DATA[719,0] := 2.59296;
   DATA[719,1] := 535.8394;
   DATA[719,2] := 2.0;
   DATA[719,3] := 2.0;
   DATA[719,4] := 262.1764;
   DATA[719,5] := 8.395475;
   DATA[719,6] := 327.7108;
   DATA[719,7] := 2.44206;
   DATA[719,8] := 2.0;
   DATA[719,9] := 2.0;
   DATA[719,10] := 2.0;
   DATA[719,11] := 3.284461;
   DATA[719,12] := 0.1743586;
   DATA[719,13] := 989.0093;
   DATA[719,14] := 1.0;
   DATA[719,15] := 1.0;
   DATA[719,16] := 1.0;
   DATA[719,17] := 1.0;
   DATA[719,18] := 1.0;
   DATA[719,19] := 1.0;
   DATA[719,20] := 148.808;
   DATA[719,21] := 155.7037;
   DATA[719,22] := 1.722872;
   DATA[719,23] := 1000.397;
   DATA[719,24] := 2.0;
   DATA[719,25] := 2.0;
   DATA[719,26] := 7.878942;
   DATA[719,27] := 144.7065;
   DATA[719,28] := 263.1056;
   DATA[719,29] := 12.11228;
   DATA[719,30] := 1.731095;
   DATA[719,31] := 1.305879;
   DATA[719,32] := 0.7352687;
   DATA[719,33] := 0.3066329;
   DATA[719,34] := 2.0;
   DATA[719,35] := 251.474;
   DATA[719,36] := 1.730048;
   DATA[719,37] := 190.1275;
   DATA[719,38] := 0.000128152;
   DATA[719,39] := 1.0;
   DATA[720,0] := 2.576306;
   DATA[720,1] := 536.0356;
   DATA[720,2] := 2.0;
   DATA[720,3] := 2.0;
   DATA[720,4] := 262.1764;
   DATA[720,5] := 8.395475;
   DATA[720,6] := 327.7108;
   DATA[720,7] := 2.44206;
   DATA[720,8] := 2.0;
   DATA[720,9] := 2.0;
   DATA[720,10] := 2.0;
   DATA[720,11] := 2.884308;
   DATA[720,12] := 0.1120968;
   DATA[720,13] := 989.0493;
   DATA[720,14] := 1.0;
   DATA[720,15] := 1.0;
   DATA[720,16] := 1.0;
   DATA[720,17] := 1.0;
   DATA[720,18] := 1.0;
   DATA[720,19] := 1.0;
   DATA[720,20] := 148.808;
   DATA[720,21] := 155.7037;
   DATA[720,22] := 1.720309;
   DATA[720,23] := 1000.205;
   DATA[720,24] := 2.0;
   DATA[720,25] := 2.0;
   DATA[720,26] := 7.878942;
   DATA[720,27] := 144.7065;
   DATA[720,28] := 263.1056;
   DATA[720,29] := 12.11228;
   DATA[720,30] := 1.732633;
   DATA[720,31] := 1.320994;
   DATA[720,32] := 0.7352687;
   DATA[720,33] := 0.3066329;
   DATA[720,34] := 2.0;
   DATA[720,35] := 251.474;
   DATA[720,36] := 1.730048;
   DATA[720,37] := 190.1275;
   DATA[720,38] := 0.000128152;
   DATA[720,39] := 1.0;
   DATA[721,0] := 2.552926;
   DATA[721,1] := 536.0749;
   DATA[721,2] := 2.0;
   DATA[721,3] := 2.0;
   DATA[721,4] := 262.1764;
   DATA[721,5] := 8.395475;
   DATA[721,6] := 327.7108;
   DATA[721,7] := 2.44206;
   DATA[721,8] := 2.0;
   DATA[721,9] := 2.0;
   DATA[721,10] := 2.0;
   DATA[721,11] := 2.29208;
   DATA[721,12] := 0.05406271;
   DATA[721,13] := 989.2496;
   DATA[721,14] := 1.0;
   DATA[721,15] := 1.0;
   DATA[721,16] := 1.0;
   DATA[721,17] := 1.0;
   DATA[721,18] := 1.0;
   DATA[721,19] := 1.0;
   DATA[721,20] := 148.808;
   DATA[721,21] := 155.7037;
   DATA[721,22] := 1.720309;
   DATA[721,23] := 1000.051;
   DATA[721,24] := 2.0;
   DATA[721,25] := 2.0;
   DATA[721,26] := 7.878942;
   DATA[721,27] := 144.7065;
   DATA[721,28] := 263.1056;
   DATA[721,29] := 12.11228;
   DATA[721,30] := 1.733145;
   DATA[721,31] := 1.321891;
   DATA[721,32] := 0.7352687;
   DATA[721,33] := 0.3066329;
   DATA[721,34] := 2.0;
   DATA[721,35] := 251.474;
   DATA[721,36] := 1.730048;
   DATA[721,37] := 190.1275;
   DATA[721,38] := 0.000128152;
   DATA[721,39] := 1.0;
   DATA[722,0] := 2.541075;
   DATA[722,1] := 536.4675;
   DATA[722,2] := 2.0;
   DATA[722,3] := 2.0;
   DATA[722,4] := 262.1764;
   DATA[722,5] := 8.395475;
   DATA[722,6] := 327.7108;
   DATA[722,7] := 2.440265;
   DATA[722,8] := 2.0;
   DATA[722,9] := 2.0;
   DATA[722,10] := 2.0;
   DATA[722,11] := 2.154427;
   DATA[722,12] := 0.02933735;
   DATA[722,13] := 989.6902;
   DATA[722,14] := 1.0;
   DATA[722,15] := 1.0;
   DATA[722,16] := 1.0;
   DATA[722,17] := 1.0;
   DATA[722,18] := 1.0;
   DATA[722,19] := 1.0;
   DATA[722,20] := 148.808;
   DATA[722,21] := 155.7037;
   DATA[722,22] := 1.720309;
   DATA[722,23] := 999.7821;
   DATA[722,24] := 2.0;
   DATA[722,25] := 2.0;
   DATA[722,26] := 7.878942;
   DATA[722,27] := 144.7065;
   DATA[722,28] := 263.1056;
   DATA[722,29] := 12.11228;
   DATA[722,30] := 1.733402;
   DATA[722,31] := 1.310363;
   DATA[722,32] := 0.7352687;
   DATA[722,33] := 0.3066329;
   DATA[722,34] := 2.0;
   DATA[722,35] := 251.474;
   DATA[722,36] := 1.730048;
   DATA[722,37] := 190.1275;
   DATA[722,38] := 0.000128152;
   DATA[722,39] := 1.0;
   DATA[723,0] := 2.521859;
   DATA[723,1] := 536.3104;
   DATA[723,2] := 2.0;
   DATA[723,3] := 2.0;
   DATA[723,4] := 262.1764;
   DATA[723,5] := 8.395475;
   DATA[723,6] := 327.7108;
   DATA[723,7] := 2.439753;
   DATA[723,8] := 2.0;
   DATA[723,9] := 2.0;
   DATA[723,10] := 2.0;
   DATA[723,11] := 2.074397;
   DATA[723,12] := 0.00192166;
   DATA[723,13] := 989.6501;
   DATA[723,14] := 1.0;
   DATA[723,15] := 1.0;
   DATA[723,16] := 1.0;
   DATA[723,17] := 1.0;
   DATA[723,18] := 1.0;
   DATA[723,19] := 1.0;
   DATA[723,20] := 148.808;
   DATA[723,21] := 155.7806;
   DATA[723,22] := 1.720309;
   DATA[723,23] := 999.7052;
   DATA[723,24] := 2.0;
   DATA[723,25] := 2.0;
   DATA[723,26] := 7.878942;
   DATA[723,27] := 144.7065;
   DATA[723,28] := 263.1056;
   DATA[723,29] := 12.11228;
   DATA[723,30] := 1.734683;
   DATA[723,31] := 1.28641;
   DATA[723,32] := 0.7352687;
   DATA[723,33] := 0.3066329;
   DATA[723,34] := 2.0;
   DATA[723,35] := 251.474;
   DATA[723,36] := 1.730048;
   DATA[723,37] := 190.1275;
   DATA[723,38] := 0.000128152;
   DATA[723,39] := 1.0;
   DATA[724,0] := 2.504244;
   DATA[724,1] := 536.2712;
   DATA[724,2] := 2.0;
   DATA[724,3] := 2.0;
   DATA[724,4] := 262.1764;
   DATA[724,5] := 8.395475;
   DATA[724,6] := 327.7108;
   DATA[724,7] := 2.439753;
   DATA[724,8] := 2.0;
   DATA[724,9] := 2.0;
   DATA[724,10] := 2.0;
   DATA[724,11] := 2.05839;
   DATA[724,13] := 990.2509;
   DATA[724,14] := 1.0;
   DATA[724,15] := 1.0;
   DATA[724,16] := 1.0;
   DATA[724,17] := 1.0;
   DATA[724,18] := 1.0;
   DATA[724,19] := 1.0;
   DATA[724,20] := 148.808;
   DATA[724,21] := 155.8318;
   DATA[724,22] := 1.720309;
   DATA[724,23] := 999.6283;
   DATA[724,24] := 2.0;
   DATA[724,25] := 2.0;
   DATA[724,26] := 7.878942;
   DATA[724,27] := 144.6039;
   DATA[724,28] := 263.1056;
   DATA[724,29] := 12.11228;
   DATA[724,30] := 1.734683;
   DATA[724,31] := 1.282567;
   DATA[724,32] := 0.7352687;
   DATA[724,33] := 0.3066329;
   DATA[724,34] := 2.0;
   DATA[724,35] := 251.474;
   DATA[724,36] := 1.730048;
   DATA[724,37] := 190.1275;
   DATA[724,38] := 0.000128152;
   DATA[724,39] := 1.0;
   DATA[725,0] := 2.485667;
   DATA[725,1] := 535.6431;
   DATA[725,2] := 2.0;
   DATA[725,3] := 2.0;
   DATA[725,4] := 262.1764;
   DATA[725,5] := 8.395475;
   DATA[725,6] := 327.6339;
   DATA[725,7] := 2.442316;
   DATA[725,8] := 2.0;
   DATA[725,9] := 2.0;
   DATA[725,10] := 2.0;
   DATA[725,11] := 2.042384;
   DATA[725,13] := 990.6514;
   DATA[725,14] := 1.0;
   DATA[725,15] := 1.0;
   DATA[725,16] := 1.0;
   DATA[725,17] := 1.0;
   DATA[725,18] := 1.0;
   DATA[725,19] := 1.0;
   DATA[725,20] := 148.808;
   DATA[725,21] := 155.8318;
   DATA[725,22] := 1.720309;
   DATA[725,23] := 999.7821;
   DATA[725,24] := 2.0;
   DATA[725,25] := 2.0;
   DATA[725,26] := 7.878942;
   DATA[725,27] := 144.6039;
   DATA[725,28] := 263.1056;
   DATA[725,29] := 12.11228;
   DATA[725,30] := 1.734683;
   DATA[725,31] := 1.295376;
   DATA[725,32] := 0.7352687;
   DATA[725,33] := 0.3066329;
   DATA[725,34] := 2.0;
   DATA[725,35] := 251.474;
   DATA[725,36] := 1.730048;
   DATA[725,37] := 190.1275;
   DATA[725,38] := 0.000128152;
   DATA[725,39] := 1.0;
   DATA[726,0] := 2.473497;
   DATA[726,1] := 535.5254;
   DATA[726,2] := 2.0;
